(* CODESYS project Core.library
   Company: _
   DefaultNamespace: Core
   Title: Core
   Placeholder: _Core
   Author: Krystian Lis et al.
   Version: 1.5.0

Project tree, tasks and I/O mapping:
  libraries: Tc2_Math, * (Beckhoff Automation GmbH); Tc2_Standard, * (Beckhoff Automation GmbH); Tc2_System, * (Beckhoff Automation GmbH); Tc2_Utilities, * (Beckhoff Automation GmbH)
  _/
    global variables Param
  Arg/
    Args/
      BOOL/
        function block BoolArg [ST]: AllowMut, BlockMut, FB_Init, Get, IsMut, OpSet, Set
        interface I_BoolArg: Get, IsMut, Set
        function IArgToIBoolArg [ST]
      DWORD/
        function block DwordArg [ST]: AllowMut, BlockMut, FB_Init, Get, IsMut, OpSet, Set
        interface I_DwordArg: Get, IsMut, Set
        function IArgToIDwordArg [ST]
      REAL/
        interface I_RealArg: Get, IsMut, Set
        function IArgToIRealtArg [ST]
        function block RealArg [ST]: AllowMut, BlockMut, FB_Init, Get, IsMut, OpSet, Set
    List/
      function block ArgList [ST]: Cap, Get, Set
      interface I_ArgList: Cap, Get
      interface I_MutArgList: Set
    Queue/
      function block ArgQueue [ST]: MutProxy, Proxy, Clear, Head, Length, List, Pop, Push, Tail
      interface I_ArgQueue: Head, Length, List, Tail
      interface I_MutArgQueue: Clear, Pop, Push
    interface I_Arg
    function IArgToIComp [ST]
    function ICompToIArg [ST]
  Broadcast/
    Helpers/
      function GetReceiver [ST]
      function GetSignal [ST]
    Receiver/
      function block AbstractReceiver [ST]: Call, Receive, Tag
      interface I_Receiver
      interface I_ReceiverNode: Receive
      function ICompToIRec [ST]
      function block Receiver [ST]: FB_init, Option, Receive, Tag
    Signal/
      interface I_Signal: Pair, Unpair
      interface I_SignalEmit: Emit, EmitTo, Option, Pair, Tag, Unpair
      interface I_SignalNode: _End, _Id, _Size, _Start
      function ICompToISignal [ST]
      function block Signal [ST]: _End, _Id, _Size, _Start, Emit, EmitTo, FB_init, Option, Pair, Proxy, Tag, Unpair
    Sys/
      Helpers/
        function _BroadcastDefragment [ST]
        function _BroadcastGetBestFit [ST]
        function _Emit [ST]
        function _Pair [ST]
        function _RegSignal [ST]
        function _Unpair [ST]
      Structs/
        data type _BroadcastStruct
        data type _BroadcastUnion
      global variables _Broadcast
  Callable/
    interface I_Callable: Call
  Dbg/
    global variables _Debug
    data type _DebugInfo
    function block DebugInfo [ST]
    function DebugMsg [ST]
    function DebugStr [ST]
    interface I_Debug
  Entity/
    Core/
      Entity/
        function block EntityEnd [ST]: FB_init
        function block EntityExtend [ST]: FB_init
        function block EntityStart [ST]: _AsIEntity, _End, _IsCompleted, _Size, _Start, Fb_init, Get, Id, Size
      function block Component [ST]: Entity, FB_init, Raw
      function GetEntity [ST]
      function GetOwnerFromRaw [ST]
      interface I_Component
      interface I_Entity
      interface I_EntityNode: _AsIEntity, _End, _IsCompleted, _Start, _Size, Get, Id, Size
      interface I_FatComponent: Entity, Raw
    List/
      function block CompList [ST]: Cap, Get, Set
      interface I_CompList: Cap, Get
      interface I_MutCompList: Set
    Set/
      function block CompSet [ST]: Append, Get
      interface I_CompSet: Append, Get
    Sys/
      _Helpers/
        function _EcDefragment [ST]
        function _EcGetBestFit [ST]
        function _EndEntity [ST]
        function _ExtendEntity [ST]
        function _RegComp [ST]
        function _StartEntity [ST]
      global variables _Ec
      data type _EcStruct
      data type _EcUnion
  Iter/
    function block Iter [ST]: FB_init, Get, Next, Peek, PeekBack, Prev, Set
  Result/
    Error/
      global variables Err
      global variables GenericResult
    function IsErr [ST]
    function IsFail [ST]
    function IsNone [ST]
    function IsOk [ST]
    function IsSome [ST]
    data type Result
    function ResultToStr [ST]
  Runtime/
    Execute/
      function block Execute [ST]: Attach, Exe, FB_init, Phase, State
      interface I_Execute: Execute
      interface I_ExecuteNode: Attach, Exe, State
    Init/
      interface I_Init: Init
      interface I_InitNode: Attach, Init, State
      function block Init [ST]: Attach, FB_init, Init, Phase, State
    global variables _Runtime
    function Runtime [ST]
  State/
    _Buffer/
      function block _StateBuffer [ST]: Length, Pop, Push
    _Machine/
      function block _StateMachine [ST]: Change, Execute, State
    Helpers/
      function GetState [ST]
      function GetStateManager [ST]
    Manager/
      interface I_StateManager: Owner, Request, Current, Pretender, Previous
      function ICompToIStateMgr [ST]
      function block StateManager [ST]: Execute, Owner, Proxy, Request, Current, Pretender, Previous
    State/
      interface I_State: Owner
      interface I_StateAdapter: _AsIStateInternal
      interface I_StateInternal: _AsIState, _InQueue, _NextInBuffer, Owner, _CanActivate, _CanDeactivate, _OnEntry, _OnExecute, _OnExit
      function ICompToIState [ST]
      function block State [ST]: _AsIState, _AsIStateInternal, _InQueue, _NextInBuffer, FB_Init, Owner, Proxy, Tag, _CanActivate, _CanDeactivate, CanActivate, CanDeactivate, _OnEntry, _OnExecute, _OnExit, OnEntry, OnExecute, OnExit
  Strings/
    Alias/
      data type Ch
      data type Str
    Strb/
      interface I_Strb: Append, FindFirstAfter, FindLastBefore, HasAfter, HasBefore, Inject, IsEmpty, Length, Prepend, Read, Remove, Set, Slice, Split
      function block Strb [ST]: _this, Append, FindFirstAfter, FindLastBefore, HasAfter, HasBefore, Inject, IsEmpty, Length, Prepend, Read, Remove, Set, Slice, Split
    Strf/
      program Strf [ST]: Fmt, Padding, SimpleTime
  Tags/
    Casts/
      function IArgToITag [ST]
      function ICompToITag [ST]
      function ICompToITagged [ST]
    Helpers/
      function GetTag [ST]
      function GetTagOption [ST]
      function HasTag [ST]
      function HasTagOption [ST]
      function MatchPath [ST]
    interface I_Tag: Id, Option
    interface I_TagCmp: AndHasOption, AndIf, HasOption, IsErr, IsFalse, IsTrue, Match, MatchId, MatchWcdId, OrIf, Set, XorIf
    interface I_Tagged: Tag
    function block Tag [ST]
    function block TagBase [ST]: FB_init, Id, Option, Proxy, Self
    function block TagCmp [ST]: _self, AndHasOption, AndIf, HasOption, IsErr, IsFalse, IsTrue, Match, MatchId, MatchWcdId, OrIf, Set, XorIf
    function block TagPath [ST]: _HasIncorrectSymbols, AddNext, AddPrev, Get, Next, Peek, PeekBack, Prev, Read, RemoveAndNext, RemoveAndPrev, Set, Swap
*)

// Broadcast/Sys/Structs/_BroadcastStruct
TYPE INTERNAL _BroadcastStruct :
STRUCT
	variant		: _BroadcastUnion;
	nType		: USINT;
END_STRUCT
END_TYPE

// Broadcast/Sys/Structs/_BroadcastUnion
TYPE INTERNAL  _BroadcastUnion :
UNION
	iSignal		: I_SignalNode;
	iReceiver	: I_ReceiverNode;
END_UNION
END_TYPE

// Dbg/_DebugInfo
TYPE INTERNAL _DebugInfo :
STRUCT
	iDebug		: I_Debug;
	sInfo		: Str;
END_STRUCT
END_TYPE

// Entity/Sys/_EcStruct
TYPE INTERNAL _EcStruct :
STRUCT
	variant		: _EcUnion;
	nType		: BYTE; // 0 - Empty, 1 - Entity, 2 - Component
END_STRUCT
END_TYPE

// Entity/Sys/_EcUnion
TYPE INTERNAL _EcUnion :
UNION
	iComponent	: I_FatComponent;
	iEntity		: I_EntityNode;
END_UNION
END_TYPE

// Result/Result
// Alias for INT values.
// | Result >= 1 - Ok/Success
// | Result = 0 - None
// | Result <=- 1 - Error
TYPE Result : INT; END_TYPE

// Strings/Alias/Ch
// Alias for STRING(1) values.
TYPE Ch : STRING(1); END_TYPE

// Strings/Alias/Str
// Alias for STRING(255) values.
TYPE Str : STRING(255); END_TYPE

// _/Param
{attribute 'qualified_only'}
// DO NOT SET ANY OF THE CAP PARAMETERS TO 0 OR LARGER THAN MAX DINT!!!
VAR_GLOBAL CONSTANT
	ENTITY_CAP		: UDINT(1..16#7FFFFFFF) := 20; // Max number of entities.
	COMP_CAP		: UDINT(1..16#7FFFFFFF) := 100; // Max number of entity-component pairings.
	
	DEBUGMSG_CAP	: UDINT(1..16#7FFFFFFF) := 10; // Max number of debug messages.
	DEBUGSTR_CAP	: UDINT(1..16#7FFFFFFF) := 500; // Max number of debug strings.
	
	SIGNAL_CAP		: UDINT(1..16#7FFFFFFF) := 20; // Max number of signals.
	RECEIVER_CAP	: UDINT(1..16#7FFFFFFF) := 100; // Max number of signal-receiver pairings.
END_VAR

// Broadcast/Sys/_Broadcast
{attribute 'qualified_only'}
VAR_GLOBAL INTERNAL
	{attribute 'ExpandFully'} 
	entry				: ARRAY[1..Param.RECEIVER_CAP] OF _BroadcastStruct;
	iSignal				: ARRAY[1..Param.SIGNAL_CAP] OF I_SignalNode;
	iFirst				: I_SignalNode;
	nRecLen				: UDINT;
	nSignalLen			: UDINT;
END_VAR

// Dbg/_Debug
{attribute 'qualified_only'}
VAR_GLOBAL INTERNAL
	debugMsg				: ARRAY[1..Param.DEBUGMSG_CAP] OF _DebugInfo;
	debugStr				: ARRAY[1..Param.DEBUGSTR_CAP] OF Str;
	
	nLastMsg				: UDINT;
	nLastStr				: UDINT;
	
	nErrorNumber			: UDINT;
END_VAR

// Entity/Sys/_Ec
// ---------------------------------------------------------------------------
// GLOBAL DATA BLOCK: _Ec
// PURPOSE:
//   This global variable block stores the primary structures for the entity-
//   component system. "iEntity" is an array of I_EntityNode, each describing
//   an entity's allocated range and metadata. "comp" is an array of ST_EcObject,
//   representing the actual slots for components or entity headers.
// ---------------------------------------------------------------------------
{attribute 'qualified_only'}
VAR_GLOBAL INTERNAL
    iEntity     : ARRAY[1..Param.ENTITY_CAP] OF I_EntityNode;   // All entity nodes
    comp        : ARRAY[1..Param.COMP_CAP] OF _EcStruct;      // Slots for components/entity headers
    
    iFirst      : I_EntityNode;  // Tracks the first (leftmost) allocated entity
    
    nEntityLen  : UDINT;         // Number of active entities
    nCompLen    : UDINT;         // Number of allocated slots in 'comp' array
	
	iUnderConstruction	: I_EntityNode; // Upon program initialization stores the entity that is being constructed.
	nConstructedScopes	: UDINT; // Keeps number of Entity scopes under construction	
END_VAR

// Result/Error/Err
{attribute 'qualified_only'}
VAR_GLOBAL CONSTANT
	Itf0			: Result := -2; // Null Interface 
	Str0			: Result := -3; // Empty String
	ItfEq			: Result := -4; // Interfaces are equal
	NoMatch			: Result := -5; // No match
	Ptr0			: Result := -6; // Null Pointer
	InvRef			: Result := -7; // Invalid reference
	Ovf				: Result := -8; // Overflow/Out of bounds
	Udf				: Result := -9; // Undefined
	Idx				: Result := -10; // Index error
	TcLib			: Result := -11; // Error caused by TwinCAT libraries
	InfLoop			: Result := -12; // Potential infinity loop
	IncArg			: Result := -13; // Incorrect input argument
	Init			: Result := -14; // Initialisation error
	NotFound		: Result := -15; // Item not found
END_VAR

// Result/Error/GenericResult
VAR_GLOBAL CONSTANT
	None	: Result := 0; // No result 
	Ok		: Result := 1; // Generic Ok
	Error	: Result := -1; // Generic Error
END_VAR

// Runtime/_Runtime
{attribute 'qualified_only'}
VAR_GLOBAL INTERNAL
	iFirstInit			: I_InitNode;
	iLastInit			: I_InitNode;

	iFirstCyclic		: I_ExecuteNode;
	iLastCyclic			: I_ExecuteNode;
	
	bInit				: BOOL := TRUE;
END_VAR

// Arg/Args/BOOL/BoolArg
(*
A broadcastable wrapper for a `BOOL` value. 
*)
FUNCTION_BLOCK BoolArg IMPLEMENTS I_BoolArg
VAR
	_val			: BOOL;
	_bMut			: BOOL := FALSE;
END_VAR

(*
Enables external modification of the internal value.
*)
METHOD AllowMut
_bMut := TRUE;
END_METHOD

(*
Disables external modification of the internal value.
*)
METHOD BlockMut
_bMut := FALSE;
END_METHOD

//FB_Init is always available implicitly and it is used primarily for initialization.
//The return value is not evaluated. For a specific influence, you can also declare the
//methods explicitly and provide additional code there with the standard initialization
//code. You can evaluate the return value.
{attribute 'hide'}
METHOD FB_Init: BOOL
VAR_INPUT
    bInitRetains: BOOL; // TRUE: the retain variables are initialized (reset warm / reset cold)
    bInCopyCode: BOOL;  // TRUE: the instance will be copied to the copy code afterward (online change)   

	initVal		: BOOL;
END_VAR
_val := initVal;
END_METHOD

(*
Reads the internal value.
*)
PROPERTY Get : BOOL
GET
Get := _val;
END_GET
END_PROPERTY

(*
Returns TRUE if the value is mutable.
*)
PROPERTY IsMut : BOOL
GET
IsMut := _bMut;
END_GET
END_PROPERTY

(*
Directly modifies the internal value, bypassing any mutability restrictions.
*)
METHOD OpSet : I_Arg
VAR_INPUT
	newVal		: BOOL;
END_VAR
_val := newVal;
OpSet := THIS^;
END_METHOD

(*
Modifies the internal value.  
Returns:
- `Ok` - Upon successful modification.
- `Error` - If mutability is disabled.
*)
METHOD Set : Result
VAR_INPUT
	newVal		: BOOL;
END_VAR
IF _bMut THEN
	_val := newVal;
	Set := Ok;
ELSE
	Set := Error;
END_IF
END_METHOD

END_FUNCTION_BLOCK

// Arg/Args/BOOL/I_BoolArg
(*
A broadcastable wrapper for a `BOOL` value. 
*)
INTERFACE I_BoolArg EXTENDS I_Arg

(*
Reads the internal value.
*)
PROPERTY Get : BOOL
GET
END_GET
END_PROPERTY

(*
Returns TRUE if the value is mutable.
*)
PROPERTY IsMut : BOOL
GET
END_GET
END_PROPERTY

(*
Modifies the internal value.  
Returns:
- `Ok` - Upon successful modification.
- `Error` - If mutability is disabled.
*)
METHOD Set : Result
VAR_INPUT
	newVal		: BOOL;
END_VAR
END_METHOD

END_INTERFACE

// Arg/I_Arg
(*
A queryable interface designed for transmitting data via a `Broadcast` system.  
Allows debugging and querying.
*)
INTERFACE I_Arg EXTENDS __SYSTEM.IQueryInterface, I_Debug

END_INTERFACE

// Dbg/I_Debug
(*
Enables a FB to be registered in the Debug table for visibility within the IDE.  
Provides no additional functionality beyond this.
*)
INTERFACE I_Debug

END_INTERFACE

// Arg/Args/BOOL/IArgToIBoolArg
(*
Casts I_Arg as I_BoolArg.
Returns:
- Ok - Success,
- Err.InvRef - Invalid reference,
- Err.Itf0 - Invalid interface,
- Err.NoMatch - Cast failed
*)
FUNCTION IArgToIBoolArg : Result
VAR_INPUT
	iIn		: I_Arg;
	iOut	: REFERENCE TO I_BoolArg;
END_VAR

IF NOT __ISVALIDREF(iOut) THEN
	IArgToIBoolArg := Err.InvRef;
	RETURN;
END_IF

IF iIn = 0 THEN
	IArgToIBoolArg := Err.Itf0;
	RETURN;
END_IF

IF __QUERYINTERFACE(iIn, iOut) THEN
	IArgToIBoolArg := Ok;
ELSE
	IArgToIBoolArg := Err.NoMatch;
END_IF

END_FUNCTION

// Arg/Args/DWORD/DwordArg
(*
A broadcastable wrapper for a `DWORD` value. 
*)
FUNCTION_BLOCK DwordArg IMPLEMENTS I_DwordArg
VAR
	_val			: DWORD;
	_bMut			: BOOL := FALSE;
END_VAR

(*
Enables external modification of the internal value.
*)
METHOD AllowMut
_bMut := TRUE;
END_METHOD

(*
Disables external modification of the internal value.
*)
METHOD BlockMut
_bMut := FALSE;
END_METHOD

//FB_Init is always available implicitly and it is used primarily for initialization.
//The return value is not evaluated. For a specific influence, you can also declare the
//methods explicitly and provide additional code there with the standard initialization
//code. You can evaluate the return value.
{attribute 'hide'}
METHOD FB_Init: BOOL
VAR_INPUT
    bInitRetains: BOOL; // TRUE: the retain variables are initialized (reset warm / reset cold)
    bInCopyCode: BOOL;  // TRUE: the instance will be copied to the copy code afterward (online change)   

	initVal		: DWORD;
END_VAR
_val := initVal;
END_METHOD

(*
Reads the internal value.
*)
PROPERTY Get : DWORD
GET
Get := _val;
END_GET
END_PROPERTY

(*
Returns TRUE if the value is mutable.
*)
PROPERTY IsMut : BOOL
GET
IsMut := _bMut;
END_GET
END_PROPERTY

(*
Directly modifies the internal value, bypassing any mutability restrictions.
*)
METHOD OpSet : I_Arg
VAR_INPUT
	newVal		: DWORD;
END_VAR
_val := newVal;
OpSet := THIS^;
END_METHOD

(*
Modifies the internal value.  
Returns:
- `Ok` - Upon successful modification.
- `Error` - If mutability is disabled.
*)
METHOD Set : Result
VAR_INPUT
	newVal		: DWORD;
END_VAR
IF _bMut THEN
	_val := newVal;
	Set := Ok;
ELSE
	Set := Error;
END_IF
END_METHOD

END_FUNCTION_BLOCK

// Arg/Args/DWORD/I_DwordArg
(*
A broadcastable wrapper for a `DWORD` value. 
*)
INTERFACE I_DwordArg EXTENDS I_Arg

(*
Reads the internal value.
*)
PROPERTY Get : DWORD
GET
END_GET
END_PROPERTY

(*
Returns TRUE if the value is mutable.
*)
PROPERTY IsMut : BOOL
GET
END_GET
END_PROPERTY

(*
Modifies the internal value.  
Returns:
- `Ok` - Upon successful modification.
- `Error` - If mutability is disabled.
*)
METHOD Set : Result
VAR_INPUT
	newVal		: DWORD;
END_VAR
END_METHOD

END_INTERFACE

// Arg/Args/DWORD/IArgToIDwordArg
(*
Casts I_Arg as I_DwordArg.
Returns:
- Ok - Success,
- Err.InvRef - Invalid reference,
- Err.Itf0 - Invalid interface,
- Err.NoMatch - Cast failed
*)
FUNCTION IArgToIDwordArg : Result
VAR_INPUT
	iIn		: I_Arg;
	iOut	: REFERENCE TO I_DwordArg;
END_VAR

IF NOT __ISVALIDREF(iOut) THEN
	IArgToIDwordArg := Err.InvRef;
	RETURN;
END_IF

IF iIn = 0 THEN
	IArgToIDwordArg := Err.Itf0;
	RETURN;
END_IF

IF __QUERYINTERFACE(iIn, iOut) THEN
	IArgToIDwordArg := Ok;
ELSE
	IArgToIDwordArg := Err.NoMatch;
END_IF

END_FUNCTION

// Arg/Args/REAL/I_RealArg
(*
A broadcastable wrapper for a `REAL` value. 
*)
INTERFACE I_RealArg EXTENDS I_Arg

(*
Reads the internal value.
*)
PROPERTY Get : REAL
GET
END_GET
END_PROPERTY

(*
Returns TRUE if the value is mutable.
*)
PROPERTY IsMut : BOOL
GET
END_GET
END_PROPERTY

(*
Modifies the internal value.  
Returns:
- `Ok` - Upon successful modification.
- `Error` - If mutability is disabled.
*)
METHOD Set : Result
VAR_INPUT
	newVal		: REAL;
END_VAR
END_METHOD

END_INTERFACE

// Arg/Args/REAL/IArgToIRealtArg
(*
Casts I_Arg as I_RealArg.
Returns:
- Ok - Success,
- Err.InvRef - Invalid reference,
- Err.Itf0 - Invalid interface,
- Err.NoMatch - Cast failed
*)
FUNCTION IArgToIRealtArg : Result
VAR_INPUT
	iIn		: I_Arg;
	iOut	: REFERENCE TO I_RealArg;
END_VAR

IF NOT __ISVALIDREF(iOut) THEN
	IArgToIRealtArg := Err.InvRef;
	RETURN;
END_IF

IF iIn = 0 THEN
	IArgToIRealtArg := Err.Itf0;
	RETURN;
END_IF

IF __QUERYINTERFACE(iIn, iOut) THEN
	IArgToIRealtArg := Ok;
ELSE
	IArgToIRealtArg := Err.NoMatch;
END_IF

END_FUNCTION

// Arg/Args/REAL/RealArg
(*
A broadcastable wrapper for a `REAL` value. 
*)
FUNCTION_BLOCK RealArg IMPLEMENTS I_RealArg
VAR
	_val			: REAL;
	_bMut			: BOOL := FALSE;
END_VAR

(*
Enables external modification of the internal value.
*)
METHOD AllowMut
_bMut := TRUE;
END_METHOD

(*
Disables external modification of the internal value.
*)
METHOD BlockMut
_bMut := FALSE;
END_METHOD

//FB_Init is always available implicitly and it is used primarily for initialization.
//The return value is not evaluated. For a specific influence, you can also declare the
//methods explicitly and provide additional code there with the standard initialization
//code. You can evaluate the return value.
{attribute 'hide'}
METHOD FB_Init: BOOL
VAR_INPUT
    bInitRetains: BOOL; // TRUE: the retain variables are initialized (reset warm / reset cold)
    bInCopyCode: BOOL;  // TRUE: the instance will be copied to the copy code afterward (online change)   

	initVal		: REAL;
END_VAR
_val := initVal;
END_METHOD

(*
Reads the internal value.
*)
PROPERTY Get : REAL
GET
Get := _val;
END_GET
END_PROPERTY

(*
Returns TRUE if the value is mutable.
*)
PROPERTY IsMut : BOOL
GET
IsMut := _bMut;
END_GET
END_PROPERTY

(*
Directly modifies the internal value, bypassing any mutability restrictions.
*)
METHOD OpSet : I_Arg
VAR_INPUT
	newVal		: REAL;
END_VAR
_val := newVal;
OpSet := THIS^;
END_METHOD

(*
Modifies the internal value.  
Returns:
- `Ok` - Upon successful modification.
- `Error` - If mutability is disabled.
*)
METHOD Set : Result
VAR_INPUT
	newVal		: REAL;
END_VAR
IF _bMut THEN
	_val := newVal;
	Set := Ok;
ELSE
	Set := Error;
END_IF
END_METHOD

END_FUNCTION_BLOCK

// Arg/List/ArgList
(*
A list implementation for managing `I_Arg`.  
*)
FUNCTION_BLOCK ArgList
VAR_GENERIC CONSTANT
	nCap	: UDINT := 100;
END_VAR

IMPLEMENTS I_MutArgList

VAR
	_iList	: ARRAY[1..nCap] OF I_Arg;
END_VAR

(*
Provides the maximum capacity of the list.
*)
PROPERTY Cap : UDINT
GET
Cap := nCap;
END_GET
END_PROPERTY

(*
Retrieves the `I_Arg` at the specified index.  
Returns:
- `Ok` - Successfully retrieves the `I_Arg`.
- `Err.Idx` - The specified index is out of bounds.
- `Err.InvRef` - Invalid output reference.
- `Err.Idx` - `iOut` = 0.
*)
METHOD Get : Result
VAR_INPUT
	nIndex		: UDINT;
	iOut		: REFERENCE TO I_Arg;
END_VAR
IF nIndex > nCap OR nIndex = 0 THEN
	Get := Err.Idx;
	RETURN;	
END_IF

IF NOT __ISVALIDREF(iOut) THEN
	Get := Err.InvRef;
	RETURN;
END_IF

iOut := _iList[nIndex];
IF iOut <> 0 THEN
	Get := Ok;
ELSE
	Get := Err.NotFound;
END_IF
END_METHOD

(*
Adds, updates, or removes an argument in the list at the specified index.  
Return:
- `Ok` - Upon successfully adding, modifying, or removing an entry.
- `Err.Idx` - When attempting to modify an entry at an out-of-bounds index.
*)
METHOD Set : Result
VAR_INPUT
	iIn		: I_Arg;
	nIndex		: UDINT;
END_VAR
IF nIndex > nCap OR nIndex = 0 THEN
	Set := Err.Idx;
	RETURN;	
END_IF

_iList[nIndex] := iIn;
Set := Ok;
END_METHOD

END_FUNCTION_BLOCK

// Arg/List/I_MutArgList
(*
A list implementation for managing `I_Arg`.  
*)
INTERFACE I_MutArgList EXTENDS I_ArgList

(*
Adds, updates, or removes an argument in the list at the specified index.  
Return:
- `Ok` - Upon successfully adding, modifying, or removing an entry.
- `Err.Idx` - When attempting to modify an entry at an out-of-bounds index.
*)
METHOD Set : Result
VAR_INPUT
	iIn		: I_Arg;
	nIndex		: UDINT;
END_VAR
END_METHOD

END_INTERFACE

// Arg/List/I_ArgList
(*
A list implementation for managing `I_Arg`.  
*)
INTERFACE I_ArgList EXTENDS I_Debug

(*
Provides the maximum capacity of the list.
*)
PROPERTY Cap : UDINT
GET
END_GET
END_PROPERTY

(*
Retrieves the `I_Arg` at the specified index.  
Returns:
- `Ok` - Successfully retrieves the `I_Arg`.
- `Err.Idx` - The specified index is out of bounds.
- `Err.InvRef` - Invalid output reference.
- `Err.Idx` - `iOut` = 0.
*)
METHOD Get : Result
VAR_INPUT
	nIndex		: UDINT;
	iOut		: REFERENCE TO I_Arg;
END_VAR
END_METHOD

END_INTERFACE

// Arg/Queue/ArgQueue
(*
A circular queue implementation for managing `I_Arg`.  
*)
FUNCTION_BLOCK ArgQueue
VAR_GENERIC CONSTANT
	nCap		: UDINT := 100;
END_VAR

IMPLEMENTS I_MutArgQueue

VAR
	_list		: ArgList<nCap>;
	_nLen		: UDINT := 0;
	_nHead		: UDINT := 1;
	_nTail		: UDINT := 1;
END_VAR

(*
Allows initializing an external interface variable with an interface pointer to this instance within declaration block.
Example:
iQueue: I_MutArgQueue;
queue: ArgQueue := (MutProxy := iQueue);
Result: iQueue <> 0 
*)
PROPERTY MutProxy : REFERENCE TO I_MutArgQueue
SET
MutProxy := THIS^;
END_SET
END_PROPERTY

(*
Allows initializing an external interface variable with an interface pointer to this instance within declaration block.
Example:
iQueue: I_ArgQueue;
queue: ArgQueue := (Proxy := iQueue);
Result: iQueue <> 0 
*)
PROPERTY Proxy : REFERENCE TO I_ArgQueue
SET
Proxy := THIS^;
END_SET
END_PROPERTY

(*
Clears the queue.
*)
METHOD Clear
_nHead := 1;
_nTail := 1;
_nLen := 0;
_list.Set(0, 1);
END_METHOD

(*
Returns the current head index of the queue, indicating the next position for insertion.
*)
PROPERTY Head : UDINT
GET
Head := _nHead;
END_GET
END_PROPERTY

PROPERTY Length : UDINT
GET
Length := _nLen;
END_GET
END_PROPERTY

(*
Provides access to the underlying list structure that holds the queue's argument objects.
*)
PROPERTY List : I_ArgList
GET
List := _list;
END_GET
END_PROPERTY

(*
Retrieves and removes the next argument from the queue.  
Advances the tail pointer, ensuring cyclic operation within the queue's capacity.
Returns:
- Ok - Returns `I_Arg`.
- Err.NotFound - Returns null, queue empty.
- Check `I_ArgList.Get` for more results.
*)
METHOD Pop : Result
VAR_INPUT
	iOut	: REFERENCE TO I_Arg;
END_VAR
IF _nLen = 0 THEN
	Pop := Err.NotFound;
	RETURN;
END_IF;

IF IsOk(_list.Get(_nHead, iOut), nOut => Pop) THEN
	_nHead := (_nHead MOD nCap) + 1;
	_nLen := _nLen - 1;
	Pop := Ok;
END_IF;
END_METHOD

(*
Adds a new argument to the queue.  
Advances the head pointer while maintaining a cyclic structure, and returns an overflow error if the queue is full.
Returns:
- Ok - Successful insertion
- Err.Ovf - Returns null, the queue is full.
- Check `I_ArgList.Set` for more results.
*)
METHOD Push : Result
VAR_INPUT
	iIn		: I_Arg;
END_VAR
IF _nLen = nCap THEN
	Push := Err.Ovf;
	RETURN;
END_IF;

IF IsOk(_list.Set(iIn, _nTail), nOut => Push) THEN
	_nTail := (_nTail MOD nCap) + 1;
	_nLen := _nLen + 1;
	Push := Ok;
END_IF;
END_METHOD

(*
Returns the current tail index of the queue, indicating the next position for retrieval.
*)
PROPERTY Tail : UDINT
GET
Tail := _nTail;
END_GET
END_PROPERTY

END_FUNCTION_BLOCK

// Arg/Queue/I_MutArgQueue
(*
A circular queue implementation for managing `I_Arg`.  
*)
INTERFACE I_MutArgQueue EXTENDS I_ArgQueue

(*
Clears the queue.
*)
METHOD Clear
END_METHOD

(*
Retrieves and removes the next argument from the queue.  
Advances the tail pointer, ensuring cyclic operation within the queue's capacity.
Returns:
- Ok - Returns `I_Arg`.
- Err.NotFound - Returns null, queue empty.
- Check `I_MutArgList.Get` for more results.
*)
METHOD Pop : Result
VAR_INPUT
	iOut	: REFERENCE TO I_Arg;
END_VAR
END_METHOD

(*
Adds a new argument to the queue.  
Advances the head pointer while maintaining a cyclic structure, and returns an overflow error if the queue is full.
Returns:
- Ok - Successful insertion.
- Err.Ovf - Returns null, the queue is full.
- Check `I_MutArgList.Set` for more results.
*)
METHOD Push : Result
VAR_INPUT
	iIn		: I_Arg;
END_VAR
END_METHOD

END_INTERFACE

// Arg/Queue/I_ArgQueue
(*
A circular queue implementation for managing `I_Arg`.  
*)
INTERFACE I_ArgQueue EXTENDS I_Debug

(*
Returns the current head index of the queue, indicating the next position for insertion.
*)
PROPERTY Head : UDINT
GET
END_GET
END_PROPERTY

PROPERTY Length : UDINT
GET
END_GET
END_PROPERTY

(*
Provides access to the underlying list structure that holds the queue's argument objects.
*)
PROPERTY List : I_ArgList
GET
END_GET
END_PROPERTY

(*
Returns the current tail index of the queue, indicating the next position for retrieval.
*)
PROPERTY Tail : UDINT
GET
END_GET
END_PROPERTY

END_INTERFACE

// Result/IsOk
// Return TRUE on a successful (Ok) result.
// Optionally carries the value over to nOut for further processing.
FUNCTION IsOk : BOOL
VAR_INPUT
    nIn : Result; // Result variable to check for success
END_VAR
VAR_OUTPUT
    nOut : Result; // Carries the input value for further use
END_VAR

IsOk := nIn > 0;
nOut := nIn;

END_FUNCTION

// Arg/IArgToIComp
(*
Casts I_Arg as I_Component.
Returns:
- Ok - Success,
- Err.InvRef - Invalid reference,
- Err.Itf0 - Invalid interface,
- Err.NoMatch - Cast failed
*)
FUNCTION IArgToIComp : Result
VAR_INPUT
	iIn		: I_Arg;
	iOut	: REFERENCE TO I_Component;
END_VAR

IF NOT __ISVALIDREF(iOut) THEN
	IArgToIComp := Err.InvRef;
	RETURN;
END_IF

IF iIn = 0 THEN
	IArgToIComp := Err.Itf0;
	RETURN;
END_IF

IF __QUERYINTERFACE(iIn, iOut) THEN
	IArgToIComp := Ok;
ELSE
	IArgToIComp := Err.NoMatch;
END_IF

END_FUNCTION

// Entity/Core/I_Component
(*
Represents a component in the Entity-Component system.  
Can be cast to other interfaces for extended functionality and interaction.
*)
INTERFACE I_Component EXTENDS __SYSTEM.IQueryInterface, I_Debug

END_INTERFACE

// Entity/Core/Component
(*
Allows registration of FB implementing `I_Component`. The framework will automatically add this function block to the entity's scope.
*)
FUNCTION_BLOCK FINAL Component IMPLEMENTS I_FatComponent
VAR
	_iComponent		: I_Component;
	_iEntity		: I_EntityNode;
END_VAR

(*
Returns parent Entity.
*)
PROPERTY Entity : I_Entity
GET
Entity := _iEntity._AsIEntity;
END_GET
END_PROPERTY

//FB_Init is always available implicitly and it is used primarily for initialization.
//The return value is not evaluated. For a specific influence, you can also declare the
//methods explicitly and provide additional code there with the standard initialization
//code. You can evaluate the return value.
{attribute 'hide'}
METHOD FB_init: BOOL
VAR_INPUT
    bInitRetains: BOOL; // TRUE: the retain variables are initialized (reset warm / reset cold)
    bInCopyCode: BOOL;  // TRUE: the instance will be copied to the copy code afterward (online change)
	
	iComponent		: I_Component;
END_VAR
VAR
	_nResult		: Result;
END_VAR
_iComponent := iComponent;
_iEntity := _Ec.iUnderConstruction;

IF _iEntity = 0 THEN
	DebugMsg(iComponent, 'Declared outside Entity scope!');
	RETURN;
END_IF
			
IF IsErr(_RegComp(_iEntity, THIS^), nOut => _nResult) THEN
	DebugMsg(iComponent, Tc2_Standard.CONCAT('Failed with code: ', ResultToStr(_nResult)));
END_IF
END_METHOD

(*
Returns raw I_Component pointer.
*)
PROPERTY Raw : I_Component
GET
Raw := _iComponent;
END_GET
END_PROPERTY

END_FUNCTION_BLOCK

// Entity/Core/I_FatComponent
(*
Stores raw I_Component value and additional metadata.
*)
INTERFACE I_FatComponent

(*
Returns parent Entity.
*)
PROPERTY Entity : I_Entity
GET
END_GET
END_PROPERTY

(*
Returns raw I_Component pointer.
*)
PROPERTY Raw : I_Component
GET
END_GET
END_PROPERTY

END_INTERFACE

// Entity/Core/I_Entity
(*
Represents a registered entity in the Entity-Component system.
*)
INTERFACE I_Entity EXTENDS I_Debug, I_EntityNode

END_INTERFACE

// Entity/Core/I_EntityNode
INTERFACE INTERNAL I_EntityNode EXTENDS I_Debug

PROPERTY INTERNAL _AsIEntity : I_Entity
GET
END_GET
END_PROPERTY

PROPERTY INTERNAL _End : UDINT
GET
END_GET
SET
END_SET
END_PROPERTY

PROPERTY INTERNAL _IsCompleted : BOOL
GET
END_GET
SET
END_SET
END_PROPERTY

PROPERTY INTERNAL _Start : UDINT
GET
END_GET
SET
END_SET
END_PROPERTY

PROPERTY INTERNAL _Size : UDINT
GET
END_GET
SET
END_SET
END_PROPERTY

(*
Retrieves a specific component from the entity based on the provided index.  
Returns `Err.NotFound` if the index is out of range or the entity size is zero.
Returns `Err.InvRef` if the reference to interface variable is invalid.
Otherwise returns `Ok`.
*)
METHOD Get : Result
VAR_INPUT
	nIndex		: UDINT;
	iOut		: REFERENCE TO I_FatComponent;
END_VAR
END_METHOD

(*
Returns the unique identifier of the entity, used for tracking and referencing within the EC system.
*)
PROPERTY Id : UDINT
GET
END_GET
END_PROPERTY

(*
Provides the size of the entity, indicating the number of components it manages.  
Note: For internal logic purposes, this value is incremented by one beyond the actual component count.
*)
PROPERTY Size : UDINT
GET
END_GET
END_PROPERTY

END_INTERFACE

// Dbg/DebugMsg
(*
Logs a debug message as a string tied to a `I_Debug` interface for inspection and troubleshooting within the IDE.
*)
FUNCTION DebugMsg
VAR_INPUT
	iDebug			: I_Debug;
	sInfo			: Str;
END_VAR

_Debug.nErrorNumber := _Debug.nErrorNumber + 1;

IF _Debug.nLastMsg < Param.DEBUGMSG_CAP THEN
	_Debug.nLastMsg := _Debug.nLastMsg + 1;
ELSE
	_Debug.nLastMsg := 1;
END_IF

_Debug.debugMsg[_Debug.nLastMsg].iDebug := iDebug;
_Debug.debugMsg[_Debug.nLastMsg].sInfo := sInfo;

END_FUNCTION

// Result/IsErr
// Return TRUE on any error value.
// Optionally carries the value over to nOut for further processing.
FUNCTION IsErr : BOOL
VAR_INPUT
    nIn : Result; // Result variable to check for an error
END_VAR
VAR_OUTPUT
    nOut : Result; // Carries the input value for further use
END_VAR

IsErr := nIn < 0;
nOut := nIn;

END_FUNCTION

// Entity/Sys/_Helpers/_RegComp
// ---------------------------------------------------------------------------
// FUNCTION:  _RegComp
// PURPOSE:   Registers a new component (iComponent) to the given entity (iEntity).
//            If the entity is new (_Start=0), attempts to allocate exactly 2 slots
//            (one for the entity header nType=1, one for the component nType=2).
//            If the entity already exists, tries to append a slot on the right
//            or shift the boundary on the left if free. If neither is possible,
//            it uses _EcGetBestFit to find a larger chunk, optionally coalescing
//            first. Finally, updates _Ec.iFirst if this entity's _Start is now
//            the leftmost among all entities.
// ---------------------------------------------------------------------------
FUNCTION INTERNAL _RegComp : Result
VAR_INPUT
    iEntity     : I_EntityNode;
    iComponent  : I_FatComponent;
END_VAR
VAR
    i           : UDINT;
    _nNextId    : UDINT;
    _nNewSize   : UDINT;
    
    _nStart     : UDINT;
    _nEnd       : UDINT;
    
    _nFirstId   : UDINT := Param.COMP_CAP;
	_nNewStart	: UDINT;
END_VAR

IF NOT _Runtime.bInit THEN
	_RegComp := Err.Init;
	RETURN;
END_IF

// Check if either iEntity or iComponent is invalid (0 indicates null).
IF iEntity = 0 OR iComponent = 0 THEN
    _RegComp := Err.Itf0;
    RETURN;
END_IF

// Check if global capacity is already at maximum.
IF _Ec.nCompLen = Param.COMP_CAP THEN
    _RegComp := Err.Ovf;
    RETURN;
END_IF

// Ensure this exact iComponent isn't already registered.
FOR i := 1 TO Param.COMP_CAP DO
    IF _Ec.comp[i].nType = 2 AND_THEN _Ec.comp[i].variant.iComponent = iComponent THEN
        _RegComp := Err.ItfEq;
        RETURN;
    END_IF
END_FOR

// If the entity is brand-new (_Start=0), try allocating exactly 2 slots.
IF iEntity._Start = 0 THEN
    CASE (_RegComp := _EcGetBestFit(2, nStart => _nStart, nEnd => _nEnd)) OF
        Ok:
            // Got a free chunk of size 2
        None:
            // No chunk found => defragment.
            CASE (_RegComp := _EcDefragment()) OF 
				Ok:
					// We can safely assume that if _EcGetBestFit and _EcDefragment didn't failed then _Ec.nCompLen + 1 is the next unoccupied slot.
					// If _EcGetBestFit failed then there is no avaliable space in the first place.
					// If _EcDefragment failed then this wouldn't be executed.
					_nStart := _Ec.nCompLen + 1;
					_nEnd := _Ec.nCompLen + 2;
				ELSE
					RETURN;
			END_CASE
        ELSE
            // If any other error, just return
            RETURN;
    END_CASE

    IF IsOk(_RegComp) THEN
        // Mark the first slot as entity header
        _Ec.comp[_nStart].nType := 1;
        _Ec.comp[_nStart].variant.iEntity := iEntity;

        // Mark the second slot as the component
        _Ec.comp[_nEnd].nType := 2;
        _Ec.comp[_nEnd].variant.iComponent := iComponent;
        
        // Update the entity’s metadata
        iEntity._Start := _nStart;
        iEntity._End   := _nEnd;
        iEntity._Size := 2;
        
        // Increase global count of used slots
        _Ec.nCompLen := _Ec.nCompLen + 2;
        
        // Update _Ec.iFirst if needed (i.e., if this is the first entity or if
        // the new entity starts to the left of the current iFirst).
        IF _Ec.iFirst = 0 THEN
            _Ec.iFirst := iEntity;
        ELSIF iEntity._Start < _Ec.iFirst._Start THEN
            _Ec.iFirst := iEntity;
        END_IF
        
        RETURN;
    ELSE
        RETURN;
    END_IF
END_IF

// Otherwise, the entity already has slots. Try extending to the right by 1 slot.
_nNextId := iEntity._End + 1;
IF _nNextId <= Param.COMP_CAP AND_THEN _Ec.comp[_nNextId].nType = 0 THEN
    // Mark that free slot as a new component
    _Ec.comp[_nNextId].nType := 2;
    _Ec.comp[_nNextId].variant.iComponent := iComponent;
    
    // Update entity info
    iEntity._End := _nNextId;
    iEntity._Size := iEntity._Size + 1;
    
    // Increase global used-slot counter
    _Ec.nCompLen := _Ec.nCompLen + 1;
    
    _RegComp := Ok;
    RETURN;
END_IF

// Try expanding to the left by shifting the boundary marker left one slot.
_nNextId := iEntity._Start - 1;
IF _nNextId > 0 AND_THEN _Ec.comp[_nNextId].nType = 0 THEN
    // Copy old boundary marker to new index
    _Ec.comp[_nNextId] := _Ec.comp[iEntity._Start];

    // Turn the old boundary marker slot into the new component
    _Ec.comp[iEntity._Start].nType := 2;
    _Ec.comp[iEntity._Start].variant.iComponent := iComponent;
    
    // Update entity to reflect new _Start
    iEntity._Start := _nNextId;
    iEntity._Size := iEntity._Size + 1;
    
    // Increase global used-slot counter
    _Ec.nCompLen := _Ec.nCompLen + 1;
    
    _RegComp := Ok;
    RETURN;
END_IF

// If neither immediate left nor right expansions are possible, we need a new chunk
_nNewSize := iEntity.Size + 1;
CASE (_RegComp := _EcGetBestFit(_nNewSize, nStart => _nStart, nEnd => _nEnd)) OF
    Ok:
        // chunk found
    None:
		// No chunk found => defragment.
		CASE (_RegComp := _EcDefragment(iEntity)) OF 
			Ok:
				// As above
				_nStart := _Ec.nCompLen + 1;
				_nEnd := _Ec.nCompLen + _nNewSize;
			ELSE
				RETURN;
		END_CASE
	Err.Ovf:
		// Check if there is enough space excluding the size of this chunk. 
		// We can do it this way as we alwyas increase chunk by 1.
		IF Param.COMP_CAP = _Ec.nCompLen THEN
			RETURN;
		END_IF
	
		CASE (_RegComp := _EcDefragment(iEntity)) OF 
			Ok:
				// As above
				_nStart := _Ec.nCompLen + 1;
				_nEnd := _Ec.nCompLen + _nNewSize;
			ELSE
				RETURN;
		END_CASE	
    ELSE
        // Other errors
        RETURN;
END_CASE

IF IsOk(_RegComp) THEN
    
    // Move the entire existing block to the new chunk
    Tc2_SYSTEM.MEMMOVE(
        ADR(_Ec.comp[_nStart]),
        ADR(_Ec.comp[iEntity._Start]),
        SIZEOF(_EcStruct) * iEntity.Size
    );

    // Clear out the old region
    Tc2_SYSTEM.MEMSET(
        ADR(_Ec.comp[iEntity._Start]),
        0,
        SIZEOF(_EcStruct) * iEntity.Size
    );
    
    // Mark the final slot in the new chunk as the new component
    _Ec.comp[_nEnd].nType := 2;
    _Ec.comp[_nEnd].variant.iComponent := iComponent;
    
    // Update the entity to reflect the new block location
    iEntity._Start := _nStart;
    iEntity._End   := _nEnd;
    iEntity._Size := _nNewSize;
    
    // One more slot used
    _Ec.nCompLen := _Ec.nCompLen + 1;
    
    // If this entity was iFirst, re-scan for the new leftmost. Otherwise,
    // if we are now to the left of iFirst, update iFirst to this entity.
    IF _Ec.iFirst = iEntity THEN
        FOR i := 1 TO _Ec.nEntityLen DO
			_nNewStart := _Ec.iEntity[i]._Start;
            IF _nNewStart <> 0 AND_THEN _nNewStart < _nFirstId THEN
                _nFirstId := _Ec.iEntity[i]._Start;
                _Ec.iFirst := _Ec.iEntity[i];
            END_IF
        END_FOR
    ELSIF iEntity._Start < _Ec.iFirst._Start THEN
        _Ec.iFirst := iEntity;
    END_IF
END_IF

END_FUNCTION

// Runtime/Init/Init
(*
Allows registration of FB implementing `I_Init`. 
*)
FUNCTION_BLOCK FINAL Init IMPLEMENTS I_InitNode, I_Debug
VAR
	_iInit			: I_Init;
	_iNext			: I_InitNode;
	_nState			: Result;
	_nPhase			: INT;
END_VAR

METHOD INTERNAL Attach : Result
VAR_INPUT
	iInit			: I_InitNode;
END_VAR
VAR
	_iThis			: I_InitNode := THIS^;
END_VAR
IF iInit = 0 THEN
	DebugMsg(0, Tc2_Standard.CONCAT(__POUNAME(), ': Itf = 0!'));
	RETURN;
END_IF

IF _iThis <> _Runtime.iLastInit THEN
	DebugMsg(THIS^, Tc2_Standard.CONCAT(__POUNAME(), ': Is not the last node!'));
	RETURN;
END_IF

IF IsSome(iInit.state) THEN
	DebugMsg(iInit, Tc2_Standard.CONCAT(__POUNAME(), ': Has already been added!'));
	RETURN;
END_IF

_Runtime.iLastInit := iInit;
_iNext := iInit;
END_METHOD

//FB_Init is always available implicitly and it is used primarily for initialization.
//The return value is not evaluated. For a specific influence, you can also declare the
//methods explicitly and provide additional code there with the standard initialization
//code. You can evaluate the return value.
{attribute 'hide'}
METHOD FB_Init: BOOL
VAR_INPUT
    bInitRetains: BOOL; // TRUE: the retain variables are initialized (reset warm / reset cold)
    bInCopyCode: BOOL;  // TRUE: the instance will be copied to the copy code afterward (online change)
	
	iInit			: I_Init;
END_VAR
IF IsSome(_nState) THEN
	RETURN;
END_IF

IF (_iInit := iInit) = 0 THEN
	_nState := Err.Itf0;
	DebugMsg(THIS^, Tc2_Standard.CONCAT(__POUNAME(), ': Itf = 0!'));
	RETURN;
END_IF



IF _Runtime.iLastInit <> 0 THEN
	IF IsErr(_Runtime.iLastInit.Attach(THIS^), nOut => _nState) THEN
		DebugMsg(THIS^, Tc2_Standard.CONCAT(__POUNAME(), ': Error Inside!'));
	END_IF
ELSE
	_Runtime.iFirstInit := THIS^;
	_Runtime.iLastInit := THIS^;
	_nState := Ok;
END_IF
END_METHOD

METHOD INTERNAL Init
VAR_INPUT
END_VAR
_iInit.Init(_nPhase);

IF _iNext <> 0 THEN
	_iNext.Init();
END_IF
END_METHOD

PROPERTY Phase : INT
GET
Phase := _nPhase;
END_GET
SET
_nPhase := Phase;
END_SET
END_PROPERTY

PROPERTY INTERNAL State : Result
GET
State := _nState;
END_GET
SET
IF IsNone(_nState) THEN
	_nState := State;
END_IF
END_SET
END_PROPERTY

END_FUNCTION_BLOCK

// Runtime/Init/I_Init
(*
A `Init` method of FB implmenting this interface will be called once upon program startup.
*)
INTERFACE I_Init EXTENDS I_Debug

(*
If registered, this method will be executed upon startup.
*)
METHOD Init
VAR_INPUT
	nPhase: INT;
END_VAR
END_METHOD

END_INTERFACE

// Runtime/Init/I_InitNode
INTERFACE INTERNAL I_InitNode EXTENDS I_Debug;

METHOD INTERNAL Attach : Result
VAR_INPUT
	iInit		: I_InitNode;
END_VAR
END_METHOD

METHOD INTERNAL Init
VAR_INPUT
END_VAR
END_METHOD

PROPERTY INTERNAL State : Result
GET
END_GET
SET
END_SET
END_PROPERTY

END_INTERFACE

// State/State/State
(*
An abstract representation of a system state, providing the foundation for implementing state-specific behavior.  
Manages its owner entity and supports state transitions within the system.  
Offers default behavior for state lifecycle methods, allowing programmers to override only the relevant parts.
*)
FUNCTION_BLOCK ABSTRACT State IMPLEMENTS I_StateInternal, I_State
VAR
	{attribute 'hide'}
	_comp						: Component(THIS^);
	{attribute 'hide'}
	_bInQueue					: BOOL;
	{attribute 'hide'}
	_iNextInBuffer				: I_StateInternal; // State Buffer management
	
	_tag			: TagBase;	
END_VAR

PROPERTY INTERNAL FINAL _AsIState : I_State
GET
_AsIState := THIS^;
END_GET
END_PROPERTY

PROPERTY INTERNAL FINAL _AsIStateInternal : I_StateInternal
GET
_AsIStateInternal := THIS^;
END_GET
END_PROPERTY

PROPERTY INTERNAL _InQueue : BOOL
GET
_InQueue := _bInQueue;
END_GET
SET
_bInQueue := _InQueue;
END_SET
END_PROPERTY

PROPERTY INTERNAL _NextInBuffer : I_StateInternal
GET
_NextInBuffer := _iNextInBuffer;
END_GET
SET
_iNextInBuffer := _NextInBuffer;
END_SET
END_PROPERTY

//FB_Init is always available implicitly and it is used primarily for initialization.
//The return value is not evaluated. For a specific influence, you can also declare the
//methods explicitly and provide additional code there with the standard initialization
//code. You can evaluate the return value.
{attribute 'hide'}
METHOD FB_Init: BOOL
VAR_INPUT
    bInitRetains: BOOL; // TRUE: the retain variables are initialized (reset warm / reset cold)
    bInCopyCode: BOOL;  // TRUE: the instance will be copied to the copy code afterward (online change)   
END_VAR
END_METHOD

(*
Returns the entity that owns this state.
*)
PROPERTY FINAL Owner : I_Entity
GET
Owner := _comp.Entity;
END_GET
END_PROPERTY

(*
Allows initializing an external interface variable with an interface pointer to this instance within declaration block.
Example:
iState: I_State;
state: SomeState := (Proxy := iState);
Result: iState <> 0 
*)
PROPERTY Proxy : REFERENCE TO I_State
SET
Proxy := THIS^;
END_SET
END_PROPERTY

(*
Provides access to the `I_Tag` associated with the state.
*)
PROPERTY FINAL Tag : I_Tag
GET
Tag := _tag;
END_GET
END_PROPERTY

METHOD INTERNAL _CanActivate : BOOL
_CanActivate := CanActivate();
END_METHOD

METHOD INTERNAL _CanDeactivate : BOOL
_CanDeactivate := CanDeactivate();
END_METHOD

(*
Determines whether the state can be activated.  
Returns `TRUE` by default but can be overridden for specific activation conditions.
*)
METHOD PROTECTED CanActivate : BOOL
VAR_INPUT
END_VAR
CanActivate := TRUE;
END_METHOD

(*
Determines whether the state can be deactivated.  
Returns `TRUE` by default but can be overridden for specific deactivation conditions.
*)
METHOD PROTECTED CanDeactivate : BOOL
VAR_INPUT
END_VAR
CanDeactivate := TRUE;
END_METHOD

METHOD INTERNAL _OnEntry
OnEntry();
END_METHOD

METHOD INTERNAL _OnExecute
OnExecute();
END_METHOD

METHOD INTERNAL _OnExit
OnExit();
END_METHOD

(*
Executed when the state is entered.  
Provides a hook for defining state-specific behavior to be performed during the transition into this state.
*)
METHOD PROTECTED OnEntry
VAR_INPUT
END_VAR
END_METHOD

(*
Executed during the state's operation.  
Used to define state-specific logic that runs while the state is active.
*)
METHOD PROTECTED OnExecute
VAR_INPUT
END_VAR
END_METHOD

(*
Executed when the state transitions to another state.  
Provides a hook for defining cleanup or transition-specific behavior.
*)
METHOD PROTECTED OnExit
VAR_INPUT
END_VAR
END_METHOD

END_FUNCTION_BLOCK

// State/State/I_StateInternal
INTERFACE INTERNAL I_StateInternal

PROPERTY INTERNAL _AsIState : I_State
GET
END_GET
END_PROPERTY

PROPERTY INTERNAL _InQueue : BOOL
GET
END_GET
SET
END_SET
END_PROPERTY

PROPERTY INTERNAL _NextInBuffer : I_StateInternal
GET
END_GET
SET
END_SET
END_PROPERTY

(*
Returns the entity that owns this state.
*)
PROPERTY Owner : I_Entity
GET
END_GET
END_PROPERTY

METHOD INTERNAL _CanActivate : BOOL
VAR_INPUT
END_VAR
END_METHOD

METHOD INTERNAL _CanDeactivate : BOOL
VAR_INPUT
END_VAR
END_METHOD

METHOD INTERNAL _OnEntry
VAR_INPUT
END_VAR
END_METHOD

METHOD INTERNAL _OnExecute
VAR_INPUT
END_VAR
END_METHOD

METHOD INTERNAL _OnExit
VAR_INPUT
END_VAR
END_METHOD

END_INTERFACE

// State/State/I_State
(*
Allows states to be cast to `I_Component`.
*)
INTERFACE I_State EXTENDS I_Tagged, I_Debug, I_StateAdapter

(*
Returns the entity that owns this state.
*)
PROPERTY Owner : I_Entity
GET
END_GET
END_PROPERTY

END_INTERFACE

// Tags/I_Tagged
(*
This component contains readable `I_Tag`.
Can be casted to `I_Component`.
*)
INTERFACE I_Tagged EXTENDS I_Component

PROPERTY Tag : I_Tag
GET
END_GET
END_PROPERTY

END_INTERFACE

// Tags/I_Tag
(*
An identifier that uses reflection to generate a unique symbol path.
It simplifies the path by removing project, PLC, and tag segments.
Can be casted to `I_Arg` and `I_Component`.
Example:
- Reflection: proj.plc.MAIN.functionBlock[*]._tag
- Path: MAIN.functionBlock.5
*)
INTERFACE I_Tag EXTENDS I_Debug, I_Component, I_Arg

// Read address path without Option segment.
PROPERTY Id : Str
GET
END_GET
END_PROPERTY

// Modify or read the optional segment.
PROPERTY Option : Str
GET
END_GET
END_PROPERTY

END_INTERFACE

// Tags/Tag
(*
An identifier that uses reflection to generate a unique symbol path.
It simplifies the path by removing project, PLC, and tag segments.
Example:
- Reflection: proj.plc.MAIN.functionBlock[*]._tag
- Path: MAIN.functionBlock.5

Tag, unlike TagBase, is a component!
*)
FUNCTION_BLOCK FINAL Tag EXTENDS TagBase
VAR
	_component		: Component(THIS^);	
END_VAR

END_FUNCTION_BLOCK

// Tags/TagBase
(*
An identifier that uses reflection to generate a unique symbol path.
It simplifies the path by removing project, PLC, and tag segments.
Example:
- Reflection: proj.plc.MAIN.functionBlock[*]._tag
- Path: MAIN.functionBlock.5

TagBase is not component!
*)
{attribute 'reflection'}
FUNCTION_BLOCK TagBase IMPLEMENTS I_Tag
VAR
	{attribute 'instance-path'} 
    {attribute 'noinit'} 
	_sId			: Str;
	_nOptionPos		: USINT;
	_nOptionLen		: USINT;
END_VAR

{attribute 'hide'}
METHOD FB_init : BOOL
VAR_INPUT
	bInitRetains : BOOL; // if TRUE, the retain variables are initialized (warm start / cold start)
	bInCopyCode : BOOL;  // if TRUE, the instance afterwards gets moved into the copy code (online change)
END_VAR
VAR
	i				: INT;
	_sChar			: Ch;
END_VAR
// Delete this name
FOR i := Tc2_Standard.LEN(_sId) TO 1 BY -1 DO
	IF Tc2_Standard.MID(_sId, 1, i) = '.' THEN
		_sId := Tc2_Standard.LEFT(_sId, i - 1);
		EXIT;
	END_IF
END_FOR

// Delete project name
FOR i := 1 TO Tc2_Standard.LEN(_sId) DO
	IF Tc2_Standard.MID(_sId, 1, i) = '.' THEN
		_sId := Tc2_Standard.DELETE(_sId, i, 1);
		EXIT;
	END_IF
END_FOR

// Delete plc name
FOR i := 1 TO Tc2_Standard.LEN(_sId) DO
	IF Tc2_Standard.MID(_sId, 1, i) = '.' THEN
		_sId := Tc2_Standard.DELETE(_sId, i, 1);
		EXIT;
	END_IF
END_FOR

// Replace '[' with '.' and remove ']' 
FOR i := 1 TO Tc2_Standard.LEN(_sId) DO
	_sChar := Tc2_Standard.MID(_sId, 1, i);
	IF _sChar = '[' THEN
		_sId := Tc2_Standard.REPLACE(_sId, '.', 1, i);
	ELSIF _sChar = ']' THEN
		_sId := Tc2_Standard.DELETE(_sId, 1, i);
	END_IF
END_FOR

_sId := Tc2_Utilities.F_ToLCase(_sID);
END_METHOD

// Read address path without Option segment.
PROPERTY Id : Str
GET
IF _nOptionPos <> 0 THEN
	Id := Tc2_Standard.DELETE(_sId, _nOptionLen + 1, _nOptionPos); 
ELSE
	Id := _sId;
END_IF
END_GET
END_PROPERTY

// Modify or read the optional segment.
PROPERTY Option : Str
GET
VAR
	i				: INT;
END_VAR
IF _nOptionPos <> 0 THEN
	Option := Tc2_Standard.DELETE(_sId, _nOptionPos, 1); 
ELSE
	Option := '';
END_IF
END_GET
SET
IF Option <> '' THEN
    _nOptionLen := INT_TO_USINT(Tc2_Standard.LEN(Option));    
    IF _nOptionPos <> 0 THEN
        _sId := Tc2_Standard.LEFT(_sId, _nOptionPos);
        _sId := Tc2_Standard.CONCAT(_sId, Option);
    ELSE
        // The option does not exist, so we append it
        _nOptionPos := INT_TO_USINT(Tc2_Standard.LEN(_sId) + 1);
        _sId := Tc2_Standard.CONCAT(_sId, '.');
        _sId := Tc2_Standard.CONCAT(_sId, Option);
    END_IF
ELSIF _nOptionPos <> 0 THEN
    _sId := Tc2_Standard.LEFT(_sId, _nOptionPos - 1);
    _nOptionPos := 0;
END_IF
END_SET
END_PROPERTY

(*
Allows initializing an external interface variable with an interface pointer to this instance within declaration block.
Example:
iTag: I_Tag;
tag: Tag := (Proxy := iTag);
Result: iTag <> 0 
*)
PROPERTY Proxy : REFERENCE TO I_Tag
SET
Proxy := THIS^;
END_SET
END_PROPERTY

// Return interface pointer to THIS^.
PROPERTY Self : I_Tag
GET
Self := THIS^;
END_GET
END_PROPERTY

END_FUNCTION_BLOCK

// State/State/I_StateAdapter
INTERFACE INTERNAL I_StateAdapter

PROPERTY INTERNAL _AsIStateInternal : I_StateInternal
GET
END_GET
END_PROPERTY

END_INTERFACE

// Result/IsSome
// Return TRUE for any value other than None (0).
// Optionally carries the value over to nOut for further processing.
FUNCTION IsSome : BOOL
VAR_INPUT
    nIn : Result; // Result variable to check for any non-None value
END_VAR
VAR_OUTPUT
    nOut : Result; // Carries the input value for further use
END_VAR

IsSome := nIn <> 0;
nOut := nIn;

END_FUNCTION

// Result/IsNone
// Return TRUE if the value is None.
// Optionally carries the value over to nOut for further processing.
FUNCTION IsNone : BOOL
VAR_INPUT
    nIn : Result; // Result variable to check for None
END_VAR
VAR_OUTPUT
    nOut : Result; // Carries the input value for further use
END_VAR

IsNone := nIn = 0;
nOut := nIn;

END_FUNCTION

// Entity/Sys/_Helpers/_EcGetBestFit
// ---------------------------------------------------------------------------
// FUNCTION:  _EcGetBestFit
// PURPOSE:   Searches the global _Ec.comp array for a contiguous block of
//            nRequiredSize free slots (nType=0). Starts searching near the
//            leftmost entity (iFirst). If found, returns Ok and sets (nStart,nEnd)
//            to the exact free range. If none found, returns None or an error.
// ---------------------------------------------------------------------------
FUNCTION INTERNAL _EcGetBestFit : Result
VAR_INPUT
    nRequiredSize	: UDINT;
END_VAR
VAR_OUTPUT
    nStart : UDINT;
    nEnd   : UDINT;
END_VAR
VAR
    _nStartIndex : UDINT;
    i            : UDINT;
    _nChunkSize  : UDINT;
END_VAR

// 1) Check if there is avaliable space for required size
IF Param.COMP_CAP - _Ec.nCompLen < nRequiredSize THEN
    _EcGetBestFit := Err.Ovf;
    RETURN;
END_IF

// 2) If there are no entities at all, the entire [1..nRequiredSize] is free.
IF _Ec.iFirst = 0 THEN
    nStart := 1;
    nEnd   := nStart + nRequiredSize - 1;
    _EcGetBestFit := Ok;
    RETURN;
END_IF

// 3) If the first entity doesn't start at index 1, we may have space
//    in [1..(_Ec.iFirst._Start - 1)], else search right after iFirst._End.
IF _Ec.iFirst._Start <> 1 THEN
    _nStartIndex := 1;
ELSE
    _nStartIndex := _Ec.iFirst._End + 1;
END_IF

// 4) Scan from _nStartIndex to the end of the comp array for free slots
FOR i := _nStartIndex TO Param.COMP_CAP DO
    
    CASE _Ec.comp[i].nType OF

        0: // FREE slot => increment the contiguous free count
            _nChunkSize := _nChunkSize + 1;

            // If we've now accumulated enough slots, return success
            IF _nChunkSize = nRequiredSize THEN
                nStart := i - _nChunkSize + 1;
                nEnd   := i;
                _EcGetBestFit := Ok;
                RETURN;
            END_IF

        1: // An entity header => skip the entire block of this entity
            _nChunkSize := 0;
            i := _Ec.comp[i].variant.iEntity._End;
            // Next iteration in the FOR loop will proceed from i+1

        ELSE // Any other nType => unexpected internal state
            _EcGetBestFit := Err.IncArg;
            RETURN;
    END_CASE
END_FOR

// 5) If we exit the loop, no suitable block was found
_EcGetBestFit := None;

END_FUNCTION

// Entity/Sys/_Helpers/_EcDefragment
// ---------------------------------------------------------------------------
// FUNCTION:  _EcCoalesce
// PURPOSE:   Compacts (coalesces) all occupied blocks in _Ec.comp[] to the
//            left, removing any gaps between them. Updates each entity's
//            _Start and _End accordingly, zeroes out remaining slots,
//            and reassigns _Ec.iFirst to the new leftmost entity, if any.
// ---------------------------------------------------------------------------
FUNCTION INTERNAL _EcDefragment : Result
VAR_INPUT
	iLastEntity		: I_EntityNode := 0;
END_VAR
VAR
	i				: UDINT;
   _temp			: ARRAY[1..Param.COMP_CAP] OF _EcStruct;
   _iSwappedEntity	: I_EntityNode;
   _nNextCopyId		: UDINT := 1;
END_VAR

// 1) If we are at maximum capacity (all slots are allocated).
IF _Ec.nCompLen = Param.COMP_CAP THEN
    _EcDefragment := Err.Ovf;
    RETURN;
END_IF

// 2) If there are no allocated slots at all, nothing to defragment.
IF _Ec.nCompLen = 0 THEN
    _EcDefragment := Ok;
    RETURN;
END_IF

// 3) We want to ensure that entity that requires more space will get it, so we move it temporarly to the end.
IF iLastEntity <> 0 THEN
	_iSwappedEntity := _Ec.iEntity[_Ec.nEntityLen];
	_Ec.iEntity[iLastEntity.Id] := _iSwappedEntity;
	_Ec.iEntity[_Ec.nEntityLen] := iLastEntity;
END_IF

// 3) Copy all chunks to the temporary table
FOR i := 1 TO _Ec.nEntityLen DO
	IF _Ec.iEntity[i]._Start <> 0 THEN
		Tc2_SYSTEM.MEMCPY(
							ADR(_temp[_nNextCopyId]),
							ADR(_Ec.comp[_Ec.iEntity[i]._Start]),
							SIZEOF(_EcStruct) * _Ec.iEntity[i].Size
						);
		_Ec.iEntity[i]._Start := _nNextCopyId;
		_nNextCopyId := _Ec.iEntity[i].Size + _nNextCopyId;
		_Ec.iEntity[i]._End := _nNextCopyId - 1;	
	END_IF
END_FOR

// 3) Move back the swapped entities, to preserve the Ids.
IF iLastEntity <> 0 THEN
	_Ec.iEntity[_iSwappedEntity.Id] := _iSwappedEntity;
	_Ec.iEntity[iLastEntity.Id] := iLastEntity;
END_IF

// 4) Copy temporary table onto the _Ec.comp table
Tc2_System.MEMCPY(
	ADR(_Ec.comp),
	ADR(_temp),
	SIZEOF(_EcStruct) * _Ec.nCompLen
);

// 5) Clear the remainging area
Tc2_System.MEMSET(
	ADR(_Ec.comp[_Ec.nCompLen + 1]),
	0,
	SIZEOF(_EcStruct) * (Param.COMP_CAP - _Ec.nCompLen)
);

// 6) First entry in _Ec.comp should always be iFirst
CASE _Ec.comp[1].nType OF
	1:
		_Ec.iFirst := _Ec.comp[1].variant.iEntity;
		_EcDefragment := Ok;
	ELSE
		_EcDefragment := Err.Udf;
END_CASE

END_FUNCTION

// Result/ResultToStr
// Converts a Result value to its corresponding string representation.
// Returns a string that describes the given Result value.
FUNCTION ResultToStr : Str
VAR_INPUT
    nResult : Result; // Result variable to convert to a string
END_VAR

CASE nResult OF
    1: ResultToStr := 'Ok';
    0: ResultToStr := 'None';
    -1: ResultToStr := 'Error';
    -2: ResultToStr := 'Itf0';
    -3: ResultToStr := 'Str0';
    -4: ResultToStr := 'ItfEq';
    -5: ResultToStr := 'NoMatch';
    -6: ResultToStr := 'Ptr0';
    -7: ResultToStr := 'InvRef';
    -8: ResultToStr := 'Ovf';
    -9: ResultToStr := 'Udf';
    -10: ResultToStr := 'Idx';
    -11: ResultToStr := 'TcLib';
    -12: ResultToStr := 'InfLoop';
    -13: ResultToStr := 'IncArg';
	-14: ResultToStr := 'Init';
	-15: ResultToStr := 'Item not found';
    ELSE
        ResultToStr := Tc2_Standard.CONCAT('Unknown result: ', INT_TO_STRING(nResult));
END_CASE

END_FUNCTION

// Arg/ICompToIArg
(*
Casts I_Component as I_Arg.
Returns:
- Ok - Success,
- Err.InvRef - Invalid reference,
- Err.Itf0 - Invalid interface,
- Err.NoMatch - Cast failed
*)
FUNCTION ICompToIArg : Result
VAR_INPUT
	iIn		: I_Component;
	iOut	: REFERENCE TO I_Arg;
END_VAR

IF NOT __ISVALIDREF(iOut) THEN
	ICompToIArg := Err.InvRef;
	RETURN;
END_IF

IF iIn = 0 THEN
	ICompToIArg := Err.Itf0;
	RETURN;
END_IF

IF __QUERYINTERFACE(iIn, iOut) THEN
	ICompToIArg := Ok;
ELSE
	ICompToIArg := Err.NoMatch;
END_IF

END_FUNCTION

// Broadcast/Helpers/GetReceiver
(*
Searches an `I_Entity` for a `I_Receiver` component matching provided id pattern.
Result:
- Ok - Returns `I_Receiver`.
- Err.NotFound - Returns null.
- Err.InvRef - Returns null.
- Err.Itf0 - Returns null, incorrect interface.
*)
FUNCTION GetReceiver : Result
VAR_INPUT
	iEntity		: I_Entity;
	sTagId		: Str;
	iOut		: REFERENCE TO I_Receiver;
END_VAR
VAR
	i			: Iter(1);
	_iComp		: I_FatComponent;
	cmp			: TagCmp;
END_VAR

IF iEntity = 0 THEN
	GetReceiver := Err.Itf0;
	RETURN;
END_IF

IF NOT __ISVALIDREF(iOut) THEN
	GetReceiver := Err.InvRef;
	RETURN;
END_IF

WHILE IsOk(iEntity.Get(i.Next(), _iComp)) DO
	IF IsOk(ICompToIRec(_iComp.Raw, iOut)) THEN
		IF cmp.Set(iOut.Tag).MatchWcdId(sTagId).IsTrue() THEN
			GetReceiver := Ok;
			RETURN;
		ELSE
			iOut := 0;
		END_IF
	END_IF
END_WHILE

END_FUNCTION

// Broadcast/Receiver/ICompToIRec
(*
Casts I_Component as I_Receiver.
Returns:
- Ok - Success,
- Err.InvRef - Invalid reference,
- Err.Itf0 - Invalid interface,
- Err.NoMatch - Cast failed
*)
FUNCTION ICompToIRec : Result
VAR_INPUT
	iIn		: I_Component;
	iOut	: REFERENCE TO I_Receiver;
END_VAR

IF NOT __ISVALIDREF(iOut) THEN
	ICompToIRec := Err.InvRef;
	RETURN;
END_IF

IF iIn = 0 THEN
	ICompToIRec := Err.Itf0;
	RETURN;
END_IF

IF __QUERYINTERFACE(iIn, iOut) THEN
	ICompToIRec := Ok;
ELSE
	ICompToIRec := Err.NoMatch;
END_IF

END_FUNCTION

// Broadcast/Receiver/I_Receiver
(*
Represents a receiver in the Broadcast system. Implements the necessary methods for receiving events and pairing signals.
Can be casted to `I_Component`.
*)
INTERFACE I_Receiver EXTENDS I_ReceiverNode, I_Tagged

END_INTERFACE

// Broadcast/Receiver/Receiver
(*
Represents a receiver in the Broadcast system. Implements the necessary methods for receiving events and pairing signals.
*)
FUNCTION_BLOCK FINAL Receiver IMPLEMENTS I_Receiver
VAR
	
	_comp			: Component(THIS^);
	_tag			: TagBase;
	_iCallable		: I_Callable;
END_VAR

//FB_Init is always available implicitly and it is used primarily for initialization.
//The return value is not evaluated. For a specific influence, you can also declare the
//methods explicitly and provide additional code there with the standard initialization
//code. You can evaluate the return value.
{attribute 'hide'}
METHOD FB_Init: BOOL
VAR_INPUT
    bInitRetains: BOOL; // TRUE: the retain variables are initialized (reset warm / reset cold)
    bInCopyCode: BOOL;  // TRUE: the instance will be copied to the copy code afterward (online change)

	iCallable	: I_Callable;
END_VAR
_iCallable := iCallable;
IF _iCallable = 0 THEN
	DebugMsg(THIS^, 'iReceiver = 0!');
END_IF
END_METHOD

(*
Allows access to Option property of the internal Tag.
*)
PROPERTY Option : Str
GET
Option := _tag.Option;
END_GET
SET
_tag.Option := Option;
END_SET
END_PROPERTY

METHOD INTERNAL Receive
VAR_INPUT
	iArg			: I_Arg;
END_VAR
IF _iCallable <> 0 THEN
	_iCallable.Call(iArg);
END_IF
END_METHOD

(*
Provides access to the tag associated with the signal.
*)
PROPERTY Tag : I_Tag
GET
Tag := _tag;
END_GET
END_PROPERTY

END_FUNCTION_BLOCK

// Callable/I_Callable
(*
An interface that represents an object callable through various systems. 
*)
INTERFACE I_Callable EXTENDS I_Debug

(*
This method provides a standardized way for other objects to interact with the object that owns it.
*)
METHOD Call
VAR_INPUT
	iArg		: I_Arg;
END_VAR
END_METHOD

END_INTERFACE

// Broadcast/Signal/Signal
(*
Represents a signal node within the Broadcast system.  
Enables the emission of events and supports pairing with receivers.
*)
FUNCTION_BLOCK FINAL Signal IMPLEMENTS I_SignalNode, I_Signal, I_SignalEmit
VAR
	_comp			: Component(THIS^);
	_tag			: TagBase;	
	_nId			: UDINT;
	_nStart			: UDINT;
	_nEnd			: UDINT;
	_nSize			: UDINT;
	_bIsLocked		: BOOL;
END_VAR

PROPERTY INTERNAL _End : UDINT
GET
_End := _nEnd;
END_GET
SET
_nEnd := _End;
END_SET
END_PROPERTY

PROPERTY INTERNAL _Id : UDINT
GET
_Id := _nId;
END_GET
END_PROPERTY

PROPERTY INTERNAL _Size : UDINT
GET
_Size := _nSize;
END_GET
SET
_nSize := _Size;
END_SET
END_PROPERTY

PROPERTY INTERNAL _Start : UDINT
GET
_Start := _nStart;
END_GET
SET
_nStart := _Start;
END_SET
END_PROPERTY

(*
Emits an argument through the signal's broadcasting system.  
If no argument is provided, it defaults to emitting the associated tag.
Returns:
- Ok - On Success
- Err.InfLoop - Upon recursive call attempt
*)
METHOD Emit : Result
VAR_INPUT
	iArg			: I_Arg := 0;
END_VAR
IF _bIsLocked THEN
	Emit := Err.InfLoop;
	RETURN;
END_IF

IF iArg = 0 THEN
	iArg := _tag;
END_IF

_bIsLocked := TRUE;
_Emit(THIS^, iArg);
_bIsLocked := FALSE;

Emit := Ok;
END_METHOD

(*
Emits an argument to a specified receiver.
Returns:
- `Ok` - If the emission is successful.
- `Err.Itf0` - If the receiver interface is invalid.
- `Err.InfLoop` - Upon recursive call attempt
*)
METHOD EmitTo : Result
VAR_INPUT
	iReceiver		: I_Receiver;
	iArg			: I_Arg := 0;
END_VAR
IF iReceiver = 0 THEN
	EmitTo := Err.Itf0;
	RETURN;
END_IF

IF _bIsLocked THEN
	EmitTo := Err.InfLoop;
	RETURN;
END_IF

IF iArg = 0 THEN
	iArg := _tag;
END_IF

_bIsLocked := TRUE;
iReceiver.Receive(iArg);
_bIsLocked := FALSE;

EmitTo := Ok;
END_METHOD

//FB_Init is always available implicitly and it is used primarily for initialization.
//The return value is not evaluated. For a specific influence, you can also declare the
//methods explicitly and provide additional code there with the standard initialization
//code. You can evaluate the return value.
{attribute 'hide'}
METHOD FB_Init: BOOL
VAR_INPUT
    bInitRetains: BOOL; // TRUE: the retain variables are initialized (reset warm / reset cold)
    bInCopyCode: BOOL;  // TRUE: the instance will be copied to the copy code afterward (online change)   
END_VAR
VAR
	_r	: Result;
END_VAR
CASE (_r := _RegSignal(THIS^, nIndex => _nId)) OF
	Ok:
		// Ignore
	Err.Ovf:
		DebugMsg(THIS^, '_Broadcast.iSignal table overflow!');
	ELSE
		DebugMsg(THIS^, TC2_Standard.CONCAT('_RefSignal(I_Signal): unknown error! Error code: ', TO_STRING(_r)));
END_CASE
END_METHOD

(*
Allows access to Option property of the internal Tag.
*)
PROPERTY Option : Str
GET
Option := _tag.Option;
END_GET
SET
_tag.Option := Option;
END_SET
END_PROPERTY

(*
Pairs the signal with a receiver.  
Returns:
- `Ok` - If pairing is successful.
- `Err.Itf0` - If the receiver interface is invalid.
- `Err.IncArg` - If the `I_Receiver` is invalid.
- `Err.ItfEq` - If the `I_Receiver` is already paired with this `I_Signal`.
- `Err.Ovf` - If there is no space for another pairing.
*)
METHOD Pair : Result
VAR_INPUT
	iReceiver		: I_Receiver;
END_VAR
IF iReceiver = 0 THEN
	Pair := Err.Itf0;
ELSE
	Pair := _Pair(THIS^, iReceiver);
END_IF
END_METHOD

(*
Allows initializing an external interface variable with an interface pointer to this instance within declaration block.
Example:
iSignal: I_Signal;
signal: Signal := (Proxy := iSignal);
Result: iSignal <> 0 
*)
PROPERTY Proxy : REFERENCE TO I_SignalEmit
SET
Proxy := THIS^;
END_SET
END_PROPERTY

(*
Provides access to the tag associated with the signal.
*)
PROPERTY Tag : I_Tag
GET
Tag := _tag;
END_GET
END_PROPERTY

(*
Unpairs the signal from a specified receiver.
Returns:
- `Ok` - If unpairing is successful.
- `Err.Itf0` - If the receiver interface is invalid.
- `Err.IncArg` - If the `I_Receiver` is invalid.
- `Err.NoMatch` - If `I_Signal` is not paired with this `I_Receiver`.
*)
METHOD Unpair : Result
VAR_INPUT
	iReceiver		: I_Receiver;
END_VAR
IF iReceiver = 0 THEN
	Unpair := Err.Itf0;
ELSE
	Unpair := _Unpair(THIS^, iReceiver);
END_IF
END_METHOD

END_FUNCTION_BLOCK

// Broadcast/Signal/I_SignalNode
INTERFACE INTERNAL I_SignalNode EXTENDS I_Debug

PROPERTY INTERNAL _End : UDINT
GET
END_GET
SET
END_SET
END_PROPERTY

PROPERTY INTERNAL _Id : UDINT
GET
END_GET
END_PROPERTY

PROPERTY INTERNAL _Size : UDINT
GET
END_GET
SET
END_SET
END_PROPERTY

PROPERTY INTERNAL _Start : UDINT
GET
END_GET
SET
END_SET
END_PROPERTY

END_INTERFACE

// Broadcast/Signal/I_Signal
(*
Enables pairing with receivers and casting to `I_Component`, but no emitting.
*)
INTERFACE I_Signal EXTENDS I_Debug, I_Tagged

(*
Pairs the signal with a receiver.  
Returns:
- `Ok` - If pairing is successful.
- `Err.Itf0` - If the receiver interface is invalid.
- `Err.IncArg` - If the `I_Receiver` is invalid.
- `Err.ItfEq` - If the `I_Receiver` is already paired with this `I_Signal`.
- `Err.Ovf` - If there is no space for another pairing.
*)
METHOD Pair : Result
VAR_INPUT
	iReceiver		: I_Receiver;
END_VAR
END_METHOD

(*
Unpairs the signal from a specified receiver.
Returns:
- `Ok` - If unpairing is successful.
- `Err.Itf0` - If the receiver interface is invalid.
- `Err.IncArg` - If the `I_Receiver` is invalid.
- `Err.NoMatch` - If `I_Signal` is not paired with this `I_Receiver`.
*)
METHOD Unpair : Result
VAR_INPUT
	iReceiver		: I_Receiver;
END_VAR
END_METHOD

END_INTERFACE

// Broadcast/Signal/I_SignalEmit
(*
Enables pairing with receivers and emitting, but not casting to `I_Component`.
*)
INTERFACE I_SignalEmit

(*
Emits an argument through the signal's broadcasting system.  
If no argument is provided, it defaults to emitting the associated tag.
Returns:
- `Ok` - On Success
- `Err.InfLoop` - Upon recursive call attempt
*)
METHOD Emit : Result
VAR_INPUT
	iArg			: I_Arg := 0;
END_VAR
END_METHOD

(*
Emits an argument to a specified receiver.
Returns:
- `Ok` - If the emission is successful.
- `Err.Itf0` - If the receiver interface is invalid.
- `Err.InfLoop` - Upon recursive call attempt
*)
METHOD EmitTo : Result
VAR_INPUT
	iReceiver		: I_Receiver;
	iArg			: I_Arg := 0;
END_VAR
END_METHOD

(*
Allows access to Option property of the internal Tag.
*)
PROPERTY Option : Str
GET
END_GET
SET
END_SET
END_PROPERTY

(*
Pairs the signal with a receiver.  
Returns:
- `Ok` - If pairing is successful.
- `Err.Itf0` - If the receiver interface is invalid.
- `Err.IncArg` - If the `I_Receiver` is invalid.
- `Err.ItfEq` - If the `I_Receiver` is already paired with this `I_Signal`.
- `Err.Ovf` - If there is no space for another pairing.
*)
METHOD Pair : Result
VAR_INPUT
	iReceiver		: I_Receiver;
END_VAR
END_METHOD

(*
Provides access to the tag associated with the signal.
*)
PROPERTY Tag : I_Tag
GET
END_GET
END_PROPERTY

(*
Unpairs the signal from a specified receiver.
Returns:
- `Ok` - If unpairing is successful.
- `Err.Itf0` - If the receiver interface is invalid.
- `Err.IncArg` - If the `I_Receiver` is invalid.
- `Err.NoMatch` - If `I_Signal` is not paired with this `I_Receiver`.
*)
METHOD Unpair : Result
VAR_INPUT
	iReceiver		: I_Receiver;
END_VAR
END_METHOD

END_INTERFACE

// Broadcast/Sys/Helpers/_Emit
FUNCTION INTERNAL _Emit : Result
VAR_INPUT
	iSignal		: I_SignalNode;
	iArg		: I_Arg;
END_VAR
VAR
	i			: UDINT;
	_nEnd		: UDINT;
END_VAR

IF iSignal = 0 THEN
	RETURN;
END_IF

IF iSignal._Start = 0 THEN
	RETURN;
END_IF

_nEnd := iSignal._End;
// Assumes that the entry table is correctly constructed which is very likely
FOR i := iSignal._Start + 1 TO _nEnd DO
	_Broadcast.entry[i].variant.iReceiver.Receive(iArg);
END_FOR

END_FUNCTION

// Broadcast/Sys/Helpers/_RegSignal
FUNCTION INTERNAL _RegSignal : Result
VAR_INPUT
    iSignal : I_SignalNode;
END_VAR
VAR_OUTPUT
	nIndex	: UDINT;
END_VAR

IF NOT _Runtime.bInit THEN
	_RegSignal := Err.Init;
	RETURN;
END_IF

IF iSignal = 0 THEN
	_RegSignal := Err.Itf0;
	RETURN;
END_IF

IF _Broadcast.nSignalLen = Param.SIGNAL_CAP THEN
	_RegSignal := Err.Ovf;
	RETURN;
END_IF

_Broadcast.nSignalLen := _Broadcast.nSignalLen + 1;
_Broadcast.iSignal[_Broadcast.nSignalLen] := iSignal;
nIndex := _Broadcast.nSignalLen;
_RegSignal := Ok;

END_FUNCTION

// Broadcast/Sys/Helpers/_Pair
FUNCTION INTERNAL _Pair : Result
VAR_INPUT
	iSignal		: I_SignalNode;
	iReceiver	: I_ReceiverNode;
END_VAR
VAR
	i			: UDINT;
	_nStart		: UDINT;
	_nEnd		: UDINT;
	_nFirstId	: UDINT;
	_nNextId	: UDINT;
	_nNewSize	: UDINT;
	_nNewStart	: UDINT;
END_VAR

// 1) Check if either iSignal or iReceiver is invalid (0 indicates null).
IF iSignal = 0 OR iReceiver = 0 THEN
	_Pair := Err.Itf0;
	RETURN;
END_IF

// 2) Check if global capacity is already at maximum.
IF _Broadcast.nRecLen = Param.RECEIVER_CAP THEN
	_Pair := Err.Ovf;
	RETURN;
END_IF

// 3) Ensure this exact iReceiver isn't already within the iSignal chunk
FOR i := iSignal._Start + 1 TO iSignal._End DO
	IF _Broadcast.entry[i].variant.iReceiver = iReceiver THEN
		_Pair := Err.ItfEq;
		RETURN;
	END_IF
END_FOR

// 4) If the signal is brand-new (_Start=0), try allocating exactly 2 slots.
IF iSignal._Start = 0 THEN
	CASE (_Pair := _BroadcastGetBestFit(2, nStart => _nStart, nEnd => _nEnd)) OF
		Ok:
			// Found a free chunk of size 2
		None:
			CASE (_Pair := _BroadcastDefragment()) OF 
				Ok:
					// We can safely assume that if _BroadcastGetBestFit and _BroadcastDefragment didn't failed then _Broadcast.nRecLen + 1 is the next unoccupied slot.
					// If _BroadcastGetBestFit failed then there is no avaliable space in the first place.
					// If _BroadcastDefragment failed then this wouldn't be executed.
					_nStart := _Broadcast.nRecLen + 1;
					_nEnd := _Broadcast.nRecLen + 2;
				ELSE
					RETURN;
			END_CASE
		ELSE
			// Any other error, just return
			RETURN;
	END_CASE

	IF IsOk(_Pair) THEN
		// Mark the first slot as signal header
		_Broadcast.entry[_nStart].nType := 1;
		_Broadcast.entry[_nStart].variant.iSignal := iSignal;

		// Mark the second slot as the receiver
		_Broadcast.entry[_nEnd].nType := 2;
		_Broadcast.entry[_nEnd].variant.iReceiver := iReceiver;

		// Update the signal's metadata
		iSignal._Start := _nStart;
		iSignal._End   := _nEnd;
		iSignal._Size := 2;

		// Increase global count of used slots
		_Broadcast.nRecLen := _Broadcast.nRecLen + 2;

		// Update _Broadcast.iFirst if needed
		IF _Broadcast.iFirst = 0 THEN
			_Broadcast.iFirst := iSignal;
		ELSIF iSignal._Start < _Broadcast.iFirst._Start THEN
			_Broadcast.iFirst := iSignal;
		END_IF

		RETURN;
	ELSE
		RETURN;
	END_IF
END_IF

// 5) If the signal already has slots, try extending to the right by 1 slot.
_nNextId := iSignal._End + 1;
IF (_nNextId <= Param.COMP_CAP) AND_THEN (_Broadcast.entry[_nNextId].nType = 0) THEN
	// Mark that free slot as a new receiver
	_Broadcast.entry[_nNextId].nType := 2;
	_Broadcast.entry[_nNextId].variant.iReceiver := iReceiver;

	// Update signal info
	iSignal._End := _nNextId;
	iSignal._Size := iSignal._Size + 1;

	// Increase global used-slot counter
	_Broadcast.nRecLen := _Broadcast.nRecLen + 1;

	_Pair := Ok;
	RETURN;
END_IF

// 6) Try expanding to the left by shifting the boundary marker left one slot.
_nNextId := iSignal._Start - 1;
IF (_nNextId > 0) AND_THEN (_Broadcast.entry[_nNextId].nType = 0) THEN
	// Copy old boundary marker to new index
	_Broadcast.entry[_nNextId] := _Broadcast.entry[iSignal._Start];

	// Turn the old boundary marker slot into the new receiver
	_Broadcast.entry[iSignal._Start].nType := 2;
	_Broadcast.entry[iSignal._Start].variant.iReceiver := iReceiver;

	// Update signal to reflect new _Start
	iSignal._Start := _nNextId;
	iSignal._Size := iSignal._Size + 1;

	// Increase global used-slot counter
	_Broadcast.nRecLen := _Broadcast.nRecLen + 1;

	_Pair := Ok;
	RETURN;
END_IF

// 7) If neither immediate left nor right expansions are possible, we need a new chunk
_nNewSize := iSignal._Size + 1;
CASE (_Pair := _BroadcastGetBestFit(_nNewSize, nStart => _nStart, nEnd => _nEnd)) OF
	Ok:
		// Chunk found
	None:
		// No chunk found => defragment.
		CASE (_Pair := _BroadcastDefragment(iSignal)) OF 
			Ok:
				// As above
				_nStart := _Broadcast.nRecLen + 1;
				_nEnd := _Broadcast.nRecLen + _nNewSize;
			ELSE
				RETURN;
		END_CASE
	ELSE
		// Other errors
		RETURN;
END_CASE

IF IsOk(_Pair) THEN

	// Move the entire existing block to the new chunk
	Tc2_SYSTEM.MEMMOVE(
		ADR(_Broadcast.entry[_nStart]),
		ADR(_Broadcast.entry[iSignal._Start]),
		SIZEOF(_BroadcastStruct) * iSignal._Size
	);

	// Clear out the old region
	Tc2_SYSTEM.MEMSET(
		ADR(_Broadcast.entry[iSignal._Start]),
		0,
		SIZEOF(_BroadcastStruct) * iSignal._Size
	);

	// Mark the final slot in the new chunk as the new receiver
	_Broadcast.entry[_nEnd].nType := 2;
	_Broadcast.entry[_nEnd].variant.iReceiver := iReceiver;

	// Update the signal to reflect the new block location
	iSignal._Start := _nStart;
	iSignal._End   := _nEnd;
	iSignal._Size := iSignal._Size + 1;

	// One more slot used
	_Broadcast.nRecLen := _Broadcast.nRecLen + 1;

	// If this signal was iFirst, re-scan for the new leftmost. 
	// Otherwise, if we are now to the left of iFirst, update iFirst.
	IF _Broadcast.iFirst = iSignal THEN
		FOR i := 1 TO _Broadcast.nSignalLen DO
			_nNewStart := _Broadcast.iSignal[i]._Start;
			IF _nNewStart <> 0 AND_THEN _nNewStart < _nFirstId THEN
				_nFirstId := _Broadcast.iSignal[i]._Start;
				_Broadcast.iFirst := _Broadcast.iSignal[i];
			END_IF
		END_FOR
	ELSIF iSignal._Start < _Broadcast.iFirst._Start THEN
		_Broadcast.iFirst := iSignal;
	END_IF
END_IF

END_FUNCTION

// Broadcast/Sys/Helpers/_BroadcastGetBestFit
FUNCTION INTERNAL _BroadcastGetBestFit : Result
VAR_INPUT
	nRequiredSize	: UDINT;
END_VAR
VAR_OUTPUT
	nStart			: UDINT;
	nEnd			: UDINT;
END_VAR
VAR
	_nStartIndex	: UDINT;
	i				: UDINT;
	_nChunkSize		: UDINT;
END_VAR

// 1) If we've already allocated the maximum number of entities, there's no space.
IF Param.RECEIVER_CAP - _Broadcast.nRecLen < nRequiredSize THEN
	_BroadcastGetBestFit := Err.Ovf;
	RETURN;
END_IF

// 2) If there are no entities at all (first-ever component),
//    just allocate from 1..(nRequiredSize).
IF _Broadcast.iFirst = 0 THEN
	nStart := 1;
	nEnd   := nStart + nRequiredSize - 1;
	_BroadcastGetBestFit := Ok;
	RETURN;
END_IF

// 3) If the first entity doesn't start at 1, we might have free space
//    in [1..(_Broadcast.iFirst._Start - 1)].
//    Otherwise, start searching right after the first entity's end.
IF _Broadcast.iFirst._Start <> 1 THEN
	_nStartIndex := 1;
ELSE
	_nStartIndex := _Broadcast.iFirst._End + 1;
END_IF

// 4) Loop from _nStartIndex to the max capacity
FOR i := _nStartIndex TO Param.RECEIVER_CAP DO

	CASE _Broadcast.entry[i].nType OF

		0: // FREE slot
			_nChunkSize := _nChunkSize + 1;

			// If we've accumulated enough contiguous slots, we're done
			IF _nChunkSize = nRequiredSize THEN
				nStart := i - _nChunkSize + 1;
				nEnd   := i;
				_BroadcastGetBestFit := Ok;
				RETURN;
			END_IF

		1: // OCCUPIED slot
			// Reset the contiguous free-space counter
			_nChunkSize := 0;

			// Jump 'i' to the last index used by this signal
			i := _Broadcast.entry[i].variant.iSignal._End;
			// The next iteration of FOR will increment 'i', continuing from (i+1)

		ELSE // Invalid slot type => internal error
			_BroadcastGetBestFit := Err.IncArg;
			RETURN;

	END_CASE

END_FOR

// 5) If we get here, no chunk of size nRequiredSize was found.
_BroadcastGetBestFit := None;

END_FUNCTION

// Broadcast/Sys/Helpers/_BroadcastDefragment
FUNCTION INTERNAL _BroadcastDefragment : Result
VAR_INPUT
	iLastSignal		: I_SignalNode := 0;
END_VAR
VAR
	i				: UDINT;
   _temp			: ARRAY[1..Param.RECEIVER_CAP] OF _BroadcastStruct;
   _iSwappedSignal	: I_SignalNode;
   _nNextCopyId		: UDINT := 1;
END_VAR

// 1) If we are at maximum capacity (all slots are allocated).
IF _Broadcast.nRecLen = Param.RECEIVER_CAP THEN
    _BroadcastDefragment := Err.Ovf;
    RETURN;
END_IF

// 2) If there are no allocated slots at all, nothing to defragment.
IF _Broadcast.nRecLen = 0 THEN
    _BroadcastDefragment := Ok;
    RETURN;
END_IF

// 3) We want to ensure that entity that requires more space will get it, so we move it temporarly to the end.
IF iLastSignal <> 0 THEN
	_iSwappedSignal := _Broadcast.iSignal[_Broadcast.nSignalLen];
	_Broadcast.iSignal[iLastSignal._Id] := _iSwappedSignal;
	_Broadcast.iSignal[_Broadcast.nSignalLen] := iLastSignal;
END_IF

// 3) Copy all chunks to the temporary table
FOR i := 1 TO _Broadcast.nSignalLen DO
	IF _Broadcast.iSignal[i]._Start <> 0 THEN
		Tc2_SYSTEM.MEMCPY(
							ADR(_temp[_nNextCopyId]),
							ADR(_Broadcast.entry[_Broadcast.iSignal[i]._Start]),
							SIZEOF(_EcStruct) * _Broadcast.iSignal[i]._Size
						);
		_Broadcast.iSignal[i]._Start := _nNextCopyId;
		_nNextCopyId := _Broadcast.iSignal[i]._Size + _nNextCopyId;
		_Broadcast.iSignal[i]._End := _nNextCopyId - 1;	
	END_IF
END_FOR

// 3) Move back the swapped entities, to preserve the Ids.
IF iLastSignal <> 0 THEN
	_Broadcast.iSignal[_iSwappedSignal._Id] := _iSwappedSignal;
	_Broadcast.iSignal[iLastSignal._Id] := iLastSignal;
END_IF

// 4) Copy temporary table onto the _Ec.comp table
Tc2_System.MEMCPY(
	ADR(_Broadcast.entry),
	ADR(_temp),
	SIZEOF(_EcStruct) * _Broadcast.nRecLen
);

// 5) Clear the remainging area
Tc2_System.MEMSET(
	ADR(_Broadcast.entry[_Broadcast.nRecLen + 1]),
	0,
	SIZEOF(_EcStruct) * (Param.RECEIVER_CAP - _Broadcast.nRecLen)
);

// 6) First entry in _Ec.comp should always be iFirst
CASE _Broadcast.entry[1].nType OF
	1:
		_BroadcastDefragment := Ok;
		_Broadcast.iFirst := _Broadcast.entry[1].variant.iSignal;
	ELSE
		_BroadcastDefragment := Err.Udf;
END_CASE

END_FUNCTION

// Broadcast/Receiver/I_ReceiverNode
INTERFACE INTERNAL I_ReceiverNode EXTENDS I_Debug

METHOD INTERNAL Receive
VAR_INPUT
	iArg			: I_Arg;
END_VAR
END_METHOD

END_INTERFACE

// Broadcast/Sys/Helpers/_Unpair
FUNCTION INTERNAL _Unpair : Result
VAR_INPUT
	iSignal		: I_SignalNode;
	iReceiver	: I_ReceiverNode;
END_VAR
VAR
	i			: UDINT;
	_nPos		: UDINT;
	_nEnd		: UDINT;
	_nFirstId	: UDINT := Param.RECEIVER_CAP;
	_nNewStart	: UDINT;
END_VAR

// 1) Basic null check
IF iSignal = 0 OR iReceiver = 0 THEN
	_Unpair := Err.Itf0;
	RETURN;
END_IF

// 2) Find iReceiver in [iSignal._Start+1 .. iSignal._End]
_nEnd := iSignal._End;
FOR i := iSignal._Start + 1 TO _nEnd DO
	IF _Broadcast.entry[i].variant.iReceiver = iReceiver THEN
		_nPos := i;
		EXIT;
	END_IF
END_FOR

// 3) If not found, return an error
IF _nPos = 0 THEN
	_Unpair := Err.NoMatch;
	RETURN;
END_IF

// 4) Decrement the signal's size (removing one receiver)
iSignal._Size := iSignal._Size - 1;

// 5) If only the header slot remains, remove the signal entirely
IF iSignal._Size = 1 THEN
	// Clear the last receiver slot
	_Broadcast.entry[_nEnd].nType := 0;
	_Broadcast.entry[_nEnd].variant.iReceiver := 0;
	// Clear the signal header slot
	_Broadcast.entry[_nEnd - 1].nType := 0;
	_Broadcast.entry[_nEnd - 1].variant.iSignal := 0;
	// Reset iSignal metadata
	iSignal._Size := 0;
	iSignal._Start := 0;
	iSignal._End := 0;

	// If this was the leftmost signal, find a new one
	IF _Broadcast.iFirst = iSignal THEN
		FOR i := 1 TO _Broadcast.nSignalLen DO
			_nNewStart := _Broadcast.iSignal[i]._Start;
			IF _nNewStart <> 0 AND_THEN _nNewStart < _nFirstId THEN
				_nFirstId := _Broadcast.iSignal[i]._Start;
				_Broadcast.iFirst := _Broadcast.iSignal[i];
			END_IF
		END_FOR
	END_IF

ELSE
	// 6) Otherwise, swap-remove from the last receiver slot
	_Broadcast.entry[_nPos] := _Broadcast.entry[_nEnd];
	iSignal._End := _nEnd - 1;
END_IF

// 7) Return success code
_Unpair := Ok;

END_FUNCTION

// Iter/Iter
// Provides iteration functionality over UDINT value.
// Requires initialization value.
FUNCTION_BLOCK FINAL Iter
VAR
	_nIter		: UDINT;
	_bFirstLoop	: BOOL := TRUE;
END_VAR

//FB_Init is always available implicitly and it is used primarily for initialization.
//The return value is not evaluated. For a specific influence, you can also declare the
//methods explicitly and provide additional code there with the standard initialization
//code. You can evaluate the return value.
{attribute 'hide'}
METHOD FB_Init: BOOL
VAR_INPUT
    bInitRetains: BOOL; // TRUE: the retain variables are initialized (reset warm / reset cold)
    bInCopyCode: BOOL;  // TRUE: the instance will be copied to the copy code afterward (online change)

	nInit		: UDINT; // Sets the initial iteration value to nInit.
END_VAR
_nIter := nInit;
END_METHOD

// Returns the current iteration value.
METHOD Get : UDINT
VAR_INPUT
END_VAR
Get := _nIter;
END_METHOD

// Increments the iteration value unless it's the first loop.
// On the first loop, returns the initial value without incrementing.
METHOD Next : UDINT
VAR_INPUT
END_VAR
IF _bFirstLoop THEN
	_bFirstLoop := FALSE;
	Next := _nIter;
	RETURN;	
END_IF

_nIter := _nIter + 1;
Next := _nIter;
END_METHOD

// Returns the next iteration value without modifying the current state.
METHOD Peek: UDINT
VAR_INPUT
END_VAR
Peek := _nIter + 1;
END_METHOD

// Returns the previous iteration value without modifying the current state.
METHOD PeekBack: UDINT
VAR_INPUT
END_VAR
PeekBack := _nIter - 1;
END_METHOD

// Decrements the iteration value unless it's the first loop.
// On the first loop, returns the initial value without decrementing.
METHOD Prev: UDINT
VAR_INPUT
END_VAR
IF _bFirstLoop THEN
	_bFirstLoop := FALSE;
	Prev := _nIter;
	RETURN;	
END_IF

_nIter := _nIter - 1;
Prev := _nIter;
END_METHOD

// Sets the iteration to a new value and resets the first loop flag.
// Returns the new value of the iteration.
METHOD Set: UDINT
VAR_INPUT
    nNewValue: UDINT; // New value to set for the iteration
END_VAR
_nIter := nNewValue;
_bFirstLoop	:= TRUE;
Set := _nIter;
END_METHOD

END_FUNCTION_BLOCK

// Tags/TagCmp
(*
A tool for performing CASE OF-like evaluations on `I_Tag`.  
It enables sequential evaluation of conditions and stops when `IsTrue`, `IsFalse`, or `IsErr` methods are invoked.
Allows method chaining.
*)
FUNCTION_BLOCK FINAL TagCmp IMPLEMENTS I_TagCmp
VAR
	_iBaseTag		: I_Tag;
	_nResult		: Result;
	_bLock			: BOOL;
END_VAR

PROPERTY PRIVATE _self : I_TagCmp
GET
VAR
	_this : I_TagCmp := THIS^;
END_VAR
_self := _this;
END_GET
END_PROPERTY

(*
Updates its internal state based on the internal status and option.  
Sets the state to `Ok` if the base tag is `Ok` and has the specified Option; otherwise, sets the state to `None`.
*)
METHOD AndHasOption : I_TagCmp

VAR_INPUT
	sOption		: Str;
END_VAR
AndHasOption := _self;
sOption := Tc2_Utilities.F_ToLCase(sOption);

IF _bLock THEN
	RETURN;
END_IF

IF _nResult = Ok AND _iBaseTag.Option = sOption THEN
	_nResult := Ok;
ELSE
	_nResult := None;
END_IF
END_METHOD

(*
Updates its internal state based on the internal status and an external condition.  
Sets the state to `Ok` if the base tag is `Ok` and the external condition is TRUE; otherwise, sets the state to `None`.
*)
METHOD AndIf : I_TagCmp
VAR_INPUT
	bCondition: BOOL;
END_VAR
AndIf := _self;

IF _bLock THEN
	RETURN;
END_IF

IF _nResult = Ok AND_THEN bCondition THEN
	_nResult := Ok;
ELSE
	_nResult := None;
END_IF
END_METHOD

(*
Updates its internal state based on the internal status and option.  
Sets the state to `Ok` if the base tag has the specified Option.
*)
METHOD HasOption : I_TagCmp
VAR_INPUT
	sOption		: Str;
END_VAR
HasOption := _self;
sOption := Tc2_Utilities.F_ToLCase(sOption);

IF _bLock THEN
	RETURN;
END_IF

CASE _nResult OF
	Ok,
	None:
		IF sOption <> '' AND_THEN _iBaseTag.Option = sOption THEN
			_nResult := Ok;
		END_IF
END_CASE
END_METHOD

(*
Returns `TRUE` if any evaluated conditions resulted in `Error`.  
Halts further evaluations by locking the current state.
*)
METHOD IsErr : BOOL
VAR_INPUT
END_VAR
IF _bLock THEN
	RETURN;
END_IF

IF _nResult >= 0 THEN
	RETURN;
END_IF

_bLock := TRUE;
IsErr := TRUE;
END_METHOD

(*
Returns `TRUE` if all evaluated conditions resulted in `FALSE`.  
Halts further evaluations by locking the current state.
*)
METHOD IsFalse : BOOL
VAR_INPUT
END_VAR
IF _bLock THEN
	RETURN;
END_IF

IF _nResult <> None THEN
	RETURN;
END_IF

_bLock := TRUE;
IsFalse := TRUE;
END_METHOD

(*
Returns `TRUE` if any evaluated condition resulted in `TRUE`.  
Halts further evaluations by locking the current state.
*)
METHOD IsTrue : BOOL
VAR_INPUT
END_VAR
IF _bLock THEN
	RETURN;
END_IF

IF _nResult <> Ok THEN
	RETURN;
END_IF

_bLock := TRUE;
IsTrue := TRUE;
END_METHOD

(*
Updates its internal state based on the internal status and external I_Tag.  
Sets the state to `Ok` if the base tag matches the external tag.
*)
METHOD Match : I_TagCmp
VAR_INPUT
	iOther: I_Tag;
END_VAR
Match := _self;

IF _bLock THEN
	RETURN;
END_IF

CASE _nResult OF
	Ok,
	None:
		IF iOther = _iBaseTag THEN
			_nResult := Ok;
		END_IF
END_CASE
END_METHOD

(*
Updates its internal state based on the internal status and a string value.  
Sets the state to `Ok` if the base tag Id matches the provided string from right to left.
*)
METHOD MatchId : I_TagCmp
VAR_INPUT
	sIdToMatch		: Str;
END_VAR
MatchId := _self;
sIdToMatch := Tc2_Utilities.F_ToLCase(sIdToMatch);

IF _bLock THEN
	RETURN;
END_IF

CASE _nResult OF
	Ok,
	None:
		IF sIdToMatch <> '' AND_THEN (Tc2_Standard.RIGHT(_iBaseTag.Id, Tc2_Standard.LEN(sIdToMatch)) = sIdToMatch) THEN
			_nResult := Ok;
		END_IF
END_CASE
END_METHOD

(*
Updates its internal state based on the internal status and a string value.  
Sets the state to `Ok` if the base tag Id matches the provided string pattern.
Allows wildcards.
*)
METHOD MatchWcdId : I_TagCmp
VAR_INPUT
	sPattern 			: Str;
END_VAR
VAR
	pttPath				: TagPath;
	pttSeg				: Str;
	pttPeek				: Str;
	addPath				: TagPath;
	addSeg				: Str;
	bMatch				: BOOL;
END_VAR
MatchWcdId := _self;

// Check lock
IF _bLock THEN
	RETURN;
END_IF

// Check result state
CASE _nResult OF
	Ok,
	None:		
		_nResult := MatchPath(_iBaseTag.Id, sPattern);
END_CASE
END_METHOD

(*
Updates its internal state based on the internal status and an external condition.  
Sets the state to `Ok` if the base tag is `Ok` or the external condition is TRUE.
*)
METHOD OrIf : I_TagCmp
VAR_INPUT
	bCondition: BOOL;
END_VAR
OrIf := _self;

IF _bLock THEN
	RETURN;
END_IF

IF _nResult = Ok OR_ELSE bCondition THEN
	_nResult := Ok;
END_IF
END_METHOD

(*
Sets a new base tag for comparison and resets the result and lock states.
Fails if `iBaseTag` is `0`;
*)
METHOD Set : I_TagCmp
VAR_INPUT
	iBaseTag	: I_Tag;
END_VAR
_iBaseTag := iBaseTag;
_nResult := None;
_bLock := FALSE;

IF iBaseTag = 0 THEN
	_nResult := Err.Itf0;
END_IF

Set := _self;
END_METHOD

(*
Updates its internal state based on the internal status and an external condition.  
Sets the state to `Ok` if the base tag is `Ok` xor the external condition is TRUE.
*)
METHOD XorIf : I_TagCmp
VAR_INPUT
	bCondition: BOOL;
END_VAR
XorIf := _self;

IF _bLock THEN
	RETURN;
END_IF

IF _nResult = Ok XOR bCondition THEN
	_nResult := Ok;
END_IF
END_METHOD

END_FUNCTION_BLOCK

// Tags/I_TagCmp
(*
A tool for performing CASE OF-like evaluations on `I_Tag`.  
It enables sequential evaluation of conditions and stops when `IsTrue`, `IsFalse`, or `IsErr` methods are invoked.
Allows method chaining.
*)
INTERFACE INTERNAL I_TagCmp

(*
Updates its internal state based on the internal status and option.  
Sets the state to `Ok` if the base tag is `Ok` and has the specified Option; otherwise, sets the state to `None`.
*)
METHOD AndHasOption : I_TagCmp
VAR_INPUT
	sOption		: Str;
END_VAR
END_METHOD

(*
Updates its internal state based on the internal status and an external condition.  
Sets the state to `Ok` if the base tag is `Ok` and the external condition is TRUE; otherwise, sets the state to `None`.
*)
METHOD AndIf : I_TagCmp
VAR_INPUT
	bCondition: BOOL;
END_VAR
END_METHOD

(*
Updates its internal state based on the internal status and option.  
Sets the state to `Ok` if the base tag has the specified Option.
*)
METHOD HasOption : I_TagCmp
VAR_INPUT
	sOption		: Str;
END_VAR
END_METHOD

(*
Returns `TRUE` if any evaluated conditions resulted in `Error`.  
Halts further evaluations by locking the current state.
*)
METHOD IsErr : BOOL
VAR_INPUT
END_VAR
END_METHOD

(*
Returns `TRUE` if all evaluated conditions resulted in `FALSE`.  
Halts further evaluations by locking the current state.
*)
METHOD IsFalse : BOOL
VAR_INPUT
END_VAR
END_METHOD

(*
Returns `TRUE` if any evaluated condition resulted in `TRUE`.  
Halts further evaluations by locking the current state.
*)
METHOD IsTrue : BOOL
VAR_INPUT
END_VAR
END_METHOD

(*
Updates its internal state based on the internal status and external I_Tag.  
Sets the state to `Ok` if the base tag matches the external tag.
*)
METHOD Match : I_TagCmp
VAR_INPUT
	iOther: I_Tag;
END_VAR
END_METHOD

(*
Updates its internal state based on the internal status and a string value.  
Sets the state to `Ok` if the base tag Id matches the provided string from right to left.
*)
METHOD MatchId : I_TagCmp
VAR_INPUT
	sIdToMatch		: Str;
END_VAR
END_METHOD

(*
Updates its internal state based on the internal status and a string value.  
Sets the state to `Ok` if the base tag Id matches the provided string pattern.
Allows wildcards.
*)
METHOD MatchWcdId : I_TagCmp
VAR_INPUT
	sPattern 			: Str;
END_VAR
END_METHOD

(*
Updates its internal state based on the internal status and an external condition.  
Sets the state to `Ok` if the base tag is `Ok` or the external condition is TRUE.
*)
METHOD OrIf : I_TagCmp
VAR_INPUT
	bCondition: BOOL;
END_VAR
END_METHOD

(*
Sets a new base tag for comparison and resets the result and lock states.
Fails if `iBaseTag` is `0`;
*)
METHOD Set : I_TagCmp
VAR_INPUT
	iBaseTag	: I_Tag;
END_VAR
END_METHOD

(*
Updates its internal state based on the internal status and an external condition.  
Sets the state to `Ok` if the base tag is `Ok` xor the external condition is TRUE.
*)
METHOD XorIf : I_TagCmp
VAR_INPUT
	bCondition: BOOL;
END_VAR
END_METHOD

END_INTERFACE

// Tags/Helpers/MatchPath
(*
Returns whether the symbol's path matches the provided pattern.
Allows wildcards in form of "*" that can cover multiple segments.
Example pattern: *.functionBlock.*.bBool
*)
FUNCTION MatchPath : Result
VAR_INPUT
    sAddress : Str;  /// The symbol's path to evaluate
    sPattern : Str;  /// The pattern to match against
END_VAR
VAR
	pttPath				: TagPath;
	pttSeg				: Str;
	pttPeek				: Str;
	addPath				: TagPath;
	addSeg				: Str;
	bMatch				: BOOL;
END_VAR

// Init
IF IsErr(addPath.Set(sAddress)) THEN
	RETURN;
END_IF
IF IsErr(pttPath.Set(sPattern)) THEN
	RETURN;
END_IF

// Advance to the next segment
WHILE IsOk(pttPath.Next(sSeg => pttSeg)) DO	
	bMatch := FALSE;
	// If the current segment is a wildcard, then peek to the next segment
	IF pttSeg = '*' THEN
		IF IsOk(pttPath.Peek(sSeg => pttPeek)) THEN
			IF pttPeek = '*' THEN
				CONTINUE; // Skip redundant wildcard if *.*.
			END_IF
		ELSE
			MatchPath := Ok;
			RETURN; // No more segments in the pattern, so it's a match as everything so far matched(.*)
		END_IF

	// If current segment is not a wildcard reset the peek.
	ELSIF pttSeg <> '*' THEN
		pttPeek := '';
	END_IF
	
	// Get the next segment of the address path
	WHILE IsOk(addPath.Next(sSeg => addSeg)) DO
		IF pttPeek <> '' THEN
			IF pttPeek = addSeg THEN
				bMatch := TRUE;
				pttPath.Next(); // Consume get next pattern segment
				EXIT;
			ELSE
				CONTINUE; // Get next address
			END_IF
		ELSIF pttSeg = addSeg THEN
			bMatch := TRUE;
			EXIT; // Consume get next pattern segment
		ELSE
			RETURN; // No match - return
		END_IF
	END_WHILE

	IF NOT bMatch THEN
		RETURN;
	END_IF

END_WHILE

IF IsOk(addPath.Peek()) THEN
	RETURN;
END_IF

MatchPath := Ok;

END_FUNCTION

// Tags/TagPath
// Manages symbols paths, supporting segment-based navigation, validation, and modification.
// Example path: MAIN.functionBlock.5.bBool
FUNCTION_BLOCK FINAL TagPath
VAR
	_sPath		: Str;
	_nLen		: INT := 0;
	_nSegStart	: INT := 0;
	_nSegEnd	: INT := 0;
END_VAR

METHOD PRIVATE _HasIncorrectSymbols : BOOL
VAR_INPUT
	sToCheck		: Str;
END_VAR
VAR
	i				: INT;
	_nStrLen		: INT := Tc2_Standard.LEN(sToCheck);
	_sChar			: Ch;
END_VAR
_sChar := Tc2_Standard.MID(sToCheck, 1, 1);
IF (_sChar >= '0') AND (_sChar <= '9') THEN
    _HasIncorrectSymbols := TRUE; // Cannot start with a number
    RETURN;
END_IF;

// Loop through the rest of the string to validate each character
FOR i := 1 TO _nStrLen DO
    _sChar := Tc2_Utilities.F_ToLCase(Tc2_Standard.MID(sToCheck, 1, i));
    
    // Check for invalid characters
    IF NOT ((_sChar >= 'a' AND _sChar <= 'z') OR 	// Lowercase letters
            (_sChar >= '0' AND _sChar <= '9') OR 	// Numbers
            (_sChar = '_') OR                 		// Underscore
			(_sChar = '*')) THEN					// Wildcard
        _HasIncorrectSymbols := TRUE; // Invalid character found
        RETURN;
    END_IF;
END_FOR;

// If no invalid characters are found, return FALSE
_HasIncorrectSymbols := FALSE;
END_METHOD

// Adds a new segment to the path after the current segment.
// Returns `Ok` if successful, `None` if invalid.
METHOD AddNext : Result
VAR_INPUT
    sToAdd : Str; // Segment to add
END_VAR
VAR
	_nNewLen	: INT := _nLen + Tc2_Standard.LEN(sToAdd) + 1;
END_VAR
IF _sPath = '' OR _nSegStart = 0 OR sToAdd = '' THEN
    AddNext := None;
    RETURN;
END_IF;

IF _HasIncorrectSymbols(sToAdd) THEN
	AddNext := None;
	RETURN;
END_IF

IF _nNewLen <= 255 THEN
	_sPath := Tc2_Standard.INSERT(_sPath, '.', _nSegEnd);
	_sPath := Tc2_Standard.INSERT(_sPath, sToAdd, _nSegEnd + 1);
	_nLen := _nNewLen;
	AddNext := Ok;
END_IF
END_METHOD

// Adds a new segment to the path before the current segment.
// Returns `Ok` if successful, `None` if invalid.
METHOD AddPrev : Result
VAR_INPUT
    sToAdd : Str; // Segment to add
END_VAR
VAR
	_nAddLen	: INT := Tc2_Standard.LEN(sToAdd);
	_nNewLen	: INT := _nLen + _nAddLen + 1;
END_VAR
IF _sPath = '' OR _nSegStart = 0 OR sToAdd = '' THEN
    AddPrev := None;
    RETURN;
END_IF;

IF _HasIncorrectSymbols(sToAdd) THEN
	AddPrev := None;
	RETURN;
END_IF

IF _nNewLen <= 255 THEN
	_sPath := Tc2_Standard.INSERT(_sPath, '.', _nSegStart - 1);
	_sPath := Tc2_Standard.INSERT(_sPath, sToAdd, _nSegStart - 2);
	_nLen := _nNewLen;
	_nSegStart := _nSegStart + _nAddLen + 1;
	_nSegEnd := _nSegEnd + _nAddLen + 1;
	AddPrev := Ok;
END_IF
END_METHOD

// Retrieves the current segment from the path.
// Returns `Ok` if successful, `None` if no segment is found.
METHOD Get : Result
VAR_OUTPUT
    sSeg : Str; // Current segment
END_VAR
IF _nSegStart = 0 THEN
	RETURN;
END_IF

sSeg := Tc2_Standard.MID(_sPath, _nSegEnd - _nSegStart + 1, _nSegStart);
IF sSeg <> '' THEN
	Get := Ok;
END_IF
END_METHOD

// Moves to the next segment in the path and retrieves it.
// Returns `Ok` if successful, `None` if no next segment exists.
METHOD Next : Result
VAR_OUTPUT
    sSeg : Str; // Next segment
END_VAR
VAR
	i			: INT;
END_VAR
// If the path is invalid or already fully processed
IF _sPath = '' OR _nSegEnd = _nLen THEN
    Next := None;
    RETURN;
END_IF;

// Initialize on the first call
IF _nSegStart = 0 THEN
    _nSegStart := 1;
    FOR i := 1 TO _nLen DO
        IF Tc2_Standard.MID(_sPath, 1, i) = '.' THEN
            _nSegEnd := i - 1;
            EXIT;
        END_IF;
    END_FOR;

	IF _nSegEnd < _nSegStart THEN
		_nSegEnd := _nLen;
	END_IF;

    sSeg := Tc2_Standard.MID(_sPath, _nSegEnd - _nSegStart + 1, _nSegStart);
    Next := Ok;
    RETURN;
END_IF;

_nSegStart := _nSegEnd + 2; // Skip the delimiter

FOR i := _nSegStart TO _nLen DO
    IF Tc2_Standard.MID(_sPath, 1, i) = '.' THEN
        _nSegEnd := i - 1;
        EXIT;
    END_IF;
END_FOR;

// If no more delimiters, this is the last segment
IF _nSegEnd < _nSegStart THEN
    _nSegEnd := _nLen;
END_IF;

sSeg := Tc2_Standard.MID(_sPath, _nSegEnd - _nSegStart + 1, _nSegStart);
Next := Ok;
END_METHOD

// Retrieves the next segment without moving the segment pointer.
// Returns Ok if successful, None if no next segment exists.
METHOD Peek : Result
VAR_OUTPUT
    sSeg : Str; // Next segment
END_VAR
VAR
	i			: INT;
	_nPeekStart	: INT := 0;
	_nPeekEnd	: INT := 0;
END_VAR
// If the path is invalid or already fully processed
IF _sPath = '' OR _nSegEnd = _nLen OR _nSegStart = 0 THEN
    Peek := None;
    RETURN;
END_IF;

_nPeekStart := _nSegEnd + 2; // Skip the delimiter

FOR i := _nPeekStart TO _nLen DO
    IF Tc2_Standard.MID(_sPath, 1, i) = '.' THEN
        _nPeekEnd := i - 1;
        EXIT;
    END_IF;
END_FOR;

// If no more delimiters, this is the last segment
IF _nPeekEnd = 0 THEN
    _nPeekEnd := _nLen;
END_IF;

sSeg := Tc2_Standard.MID(_sPath, _nPeekEnd - _nPeekStart + 1, _nPeekStart);
Peek := Ok;
END_METHOD

// Retrieves the previous segment without moving the segment pointer.
// Returns `Ok` if successful, `None` if no previous segment exists.
METHOD PeekBack : Result
VAR_OUTPUT
    sSeg : Str; // Previous segment
END_VAR
VAR
	i			: INT;
	_nPeekStart	: INT := 0;
	_nPeekEnd	: INT := 0;
END_VAR
// If the path is invalid or already fully processed
IF _sPath = '' OR _nSegEnd = 0 OR _nSegStart = 1 THEN
    PeekBack := None;
    RETURN;
END_IF;

_nPeekEnd := _nSegStart - 2; // Skip the delimiter

FOR i := _nPeekEnd TO 1 BY -1 DO
    IF Tc2_Standard.MID(_sPath, 1, i) = '.' THEN
        _nPeekStart := i + 1;
        EXIT;
    END_IF;
END_FOR;

// If no more delimiters, this is the first segment
IF _nPeekStart = 0 THEN
    _nPeekStart := 1;
END_IF;

sSeg := Tc2_Standard.MID(_sPath, _nPeekEnd - _nPeekStart + 1, _nPeekStart);
PeekBack := Ok;
END_METHOD

// Moves to the previous segment in the path and retrieves it.
// Returns `Ok` if successful, `None` if no previous segment exists.
METHOD Prev : Result
VAR_OUTPUT
    sSeg : Str; // Previous segment
END_VAR
VAR
	i			: INT;
END_VAR
// If the path is invalid or already fully processed
IF _sPath = '' OR _nSegStart = 1 THEN
    Prev := None;
    RETURN;
END_IF;

// Initialize on the first call
IF _nSegEnd = 0 THEN
    _nSegEnd := _nLen;
    FOR i := _nSegEnd TO 1 BY -1 DO
        IF Tc2_Standard.MID(_sPath, 1, i) = '.' THEN
            _nSegStart := i + 1;
            EXIT;
        END_IF;
    END_FOR;

	// If no more delimiters, this is the first segment
	IF _nSegEnd < _nSegStart THEN
		_nSegStart := 1;
	END_IF;

    sSeg := Tc2_Standard.MID(_sPath, _nSegEnd - _nSegStart + 1, _nSegStart);
    Prev := Ok;
    RETURN;
END_IF;

_nSegEnd := _nSegStart - 2; // Skip the delimiter

FOR i := _nSegEnd TO 1 BY -1 DO
    IF Tc2_Standard.MID(_sPath, 1, i) = '.' THEN
        _nSegStart := i + 1;
        EXIT;
    END_IF;
END_FOR;

// If no more delimiters, this is the first segment
IF _nSegEnd < _nSegStart THEN
    _nSegStart := 1;
END_IF;

sSeg := Tc2_Standard.MID(_sPath, _nSegEnd - _nSegStart + 1, _nSegStart);
Prev := Ok;
END_METHOD

// Reads and returns the entire symbolic path as a string.
METHOD Read : Str
Read := _sPath;
END_METHOD

// Removes the current segment and moves to the next segment.
// Returns `Ok` if successful, `None` if no segment to remove.
METHOD RemoveAndNext : Result
VAR
    _nSegLen		: INT := _nSegEnd - _nSegStart + 1; // Length of the segment to remove
    _bIsFirstSeg	: BOOL := (_nSegStart = 1); // Check if the segment is the first segment
    _bIsLastSeg		: BOOL := (_nSegEnd = _nLen); // Check if the segment is the last segment
	i				: INT;
END_VAR
// Ensure the current path is valid
IF _sPath = '' OR _nSegStart = 0 THEN
    RemoveAndNext := None;
    RETURN;
END_IF;

